(* Logix 5000 project; controller ABB_Drive_Test vendor 1 type 14 code 149 rev 33.12; software revision 33.01; part 5 of 6 *)
(* tags used below, declared in another part *)
   ad_pointer : DINT;
   cf_bigWcmd01 : DINT;
   cf_bigWoffset01 : DINT;
   cfbw01 : CF_big_write;
   check_log_age : BOOL;
   d1hf_copy : BOOL;
   DataIndex : DINT;
   dayms_frac : REAL;
   daysince1900 : DINT;
   daysinprevmonths : DINT[13];
   detect_1st_half_full : BOOL;
   filename : STRING;
   filename_end : STRING;
   filenamestart : STRING;
   ldt : DateTime;
   log_check_active : BOOL;
   logfile_size : DINT;
   logging_enabled : BOOL;   // HABILITAR DATALOGGER
   logpulse : BOOL;
   max_file_size : DINT;
   max_logfiles : DINT;
   nr_of_writes : DINT;
   sec_pulse : TIMER;
   tempstring : STRING;
   tmpDINT : DINT;
   trigger_write : BOOL;
   write_1st_half : BOOL;
   write_length : DINT;
   write_offset : DINT;
   wrSEQ : DINT;
   Year_1901 : DINT;
   asciidata : SINT[11000];
   CF_RW_functions : CF_functions;
   manual_log_trigger : BOOL;
   SrcData : REAL[10];
(* CSVProgram, continued *)

ROUTINE MainRoutine   (* ladder *)
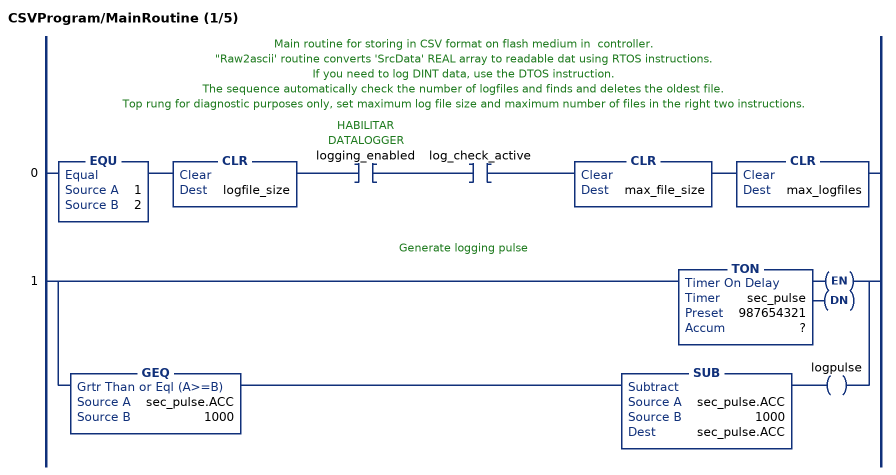
   // Main routine for storing in CSV format on flash medium in  controller.
   // "Raw2ascii' routine converts 'SrcData' REAL array to readable dat using RTOS instructions.
   // If you need to log DINT data, use the DTOS instruction.
   // The sequence automatically check the number of logfiles and finds and deletes the oldest file.
   // Top rung for diagnostic purposes only, set maximum log file size and maximum number of files in the right two instructions.
   0: EQU(1,2)CLR(logfile_size)XIC(logging_enabled)XIC(log_check_active)CLR(max_file_size)CLR(max_logfiles);
   // Generate logging pulse
   1: [TON(sec_pulse,?,?) ,GEQ(sec_pulse.ACC,1000) SUB(sec_pulse.ACC,1000,sec_pulse.ACC) OTE(logpulse) ];
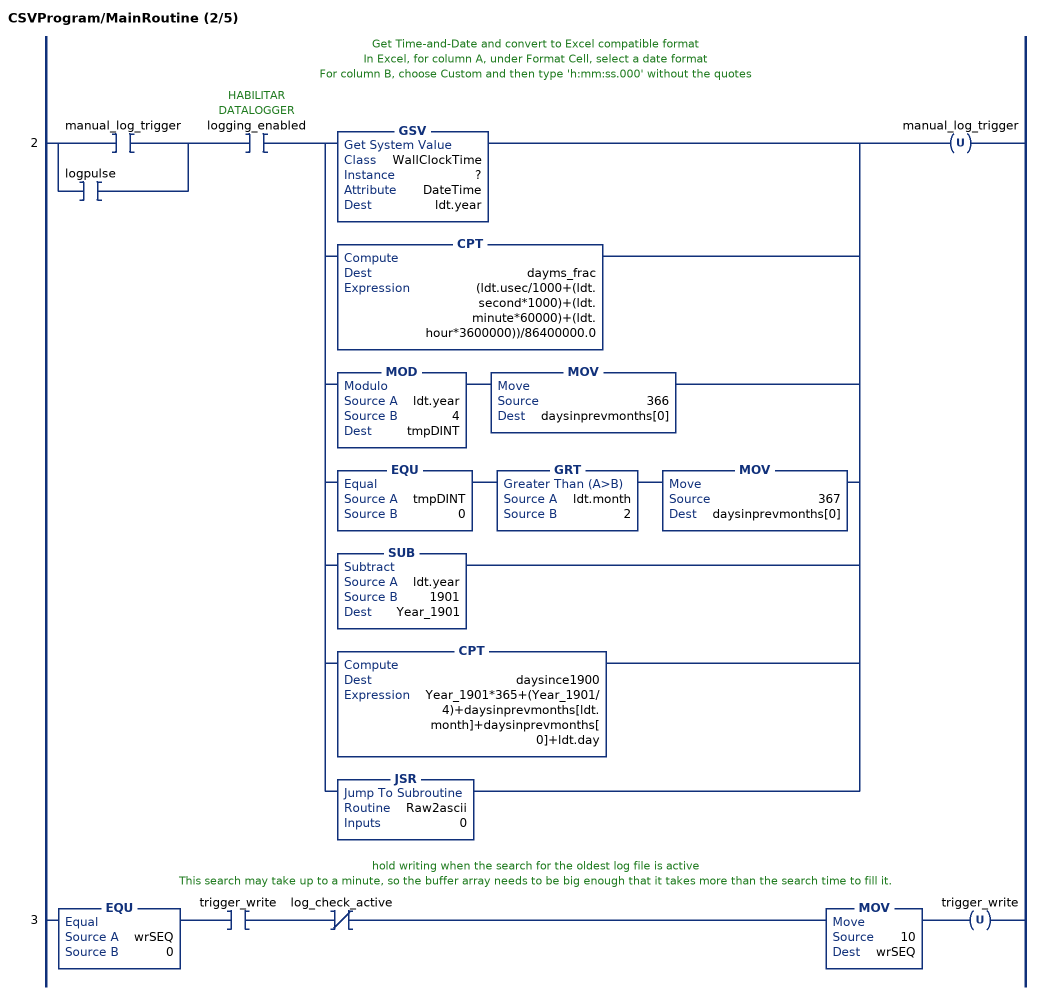
   // Get Time-and-Date and convert to Excel compatible format
   // In Excel, for column A, under Format Cell, select a date format
   // For column B, choose Custom and then type 'h:mm:ss.000' without the quotes
   2: [XIC(manual_log_trigger) ,XIC(logpulse) ]XIC(logging_enabled)[GSV(WallClockTime,?,DateTime,ldt.year) ,CPT(dayms_frac,(ldt.usec/1000+(ldt.second*1000)+(ldt.minute*60000)+(ldt.hour*3600000))/86400000.0) ,MOD(ldt.year,4,tmpDINT) MOV(366,daysinprevmonths[0]) ,EQU(tmpDINT,0) GRT(ldt.month,2) MOV(367,daysinprevmonths[0]) ,SUB(ldt.year,1901,Year_1901) ,CPT(daysince1900,Year_1901*365+(Year_1901/4)+daysinprevmonths[ldt.month]+daysinprevmonths[0]+ldt.day) ,JSR(Raw2ascii,0) ]OTU(manual_log_trigger);
   // hold writing when the search for the oldest log file is active
   // This search may take up to a minute, so the buffer array needs to be big enough that it takes more than the search time to fill it.
   3: EQU(wrSEQ,0)XIC(trigger_write)XIO(log_check_active)MOV(10,wrSEQ)OTU(trigger_write);
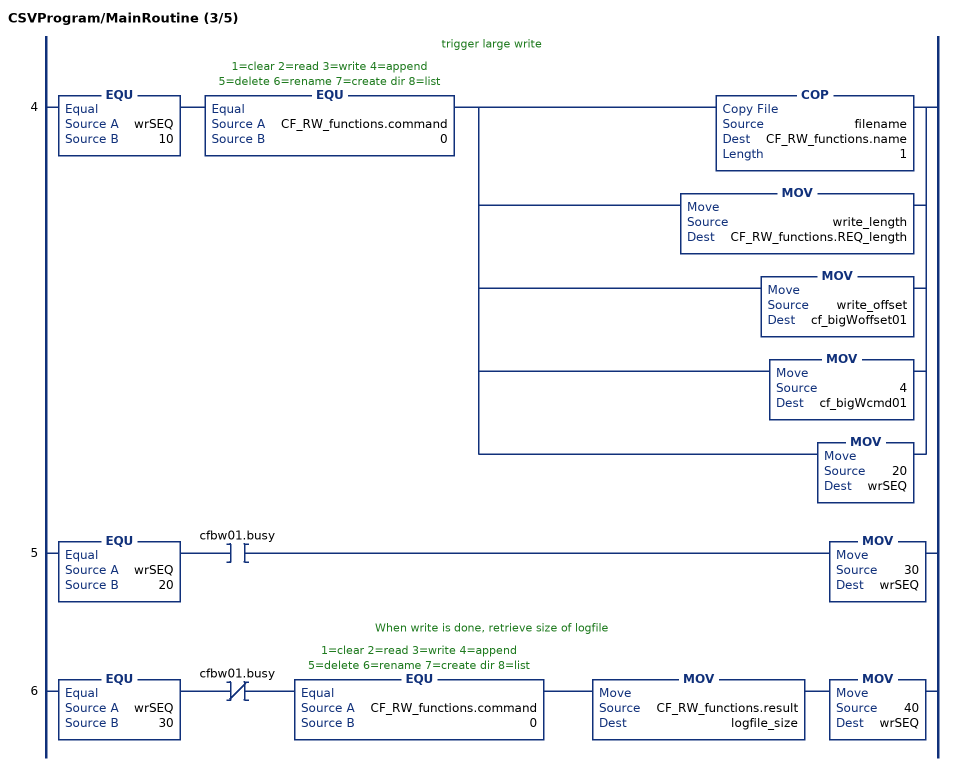
   // trigger large write
   4: EQU(wrSEQ,10)EQU(CF_RW_functions.command,0)[COP(filename,CF_RW_functions.name,1) ,MOV(write_length,CF_RW_functions.REQ_length) ,MOV(write_offset,cf_bigWoffset01) ,MOV(4,cf_bigWcmd01) ,MOV(20,wrSEQ) ];
   5: EQU(wrSEQ,20)XIC(cfbw01.busy)MOV(30,wrSEQ);
   // When write is done, retrieve size of logfile
   6: EQU(wrSEQ,30)XIO(cfbw01.busy)EQU(CF_RW_functions.command,0)MOV(CF_RW_functions.result,logfile_size)MOV(40,wrSEQ);
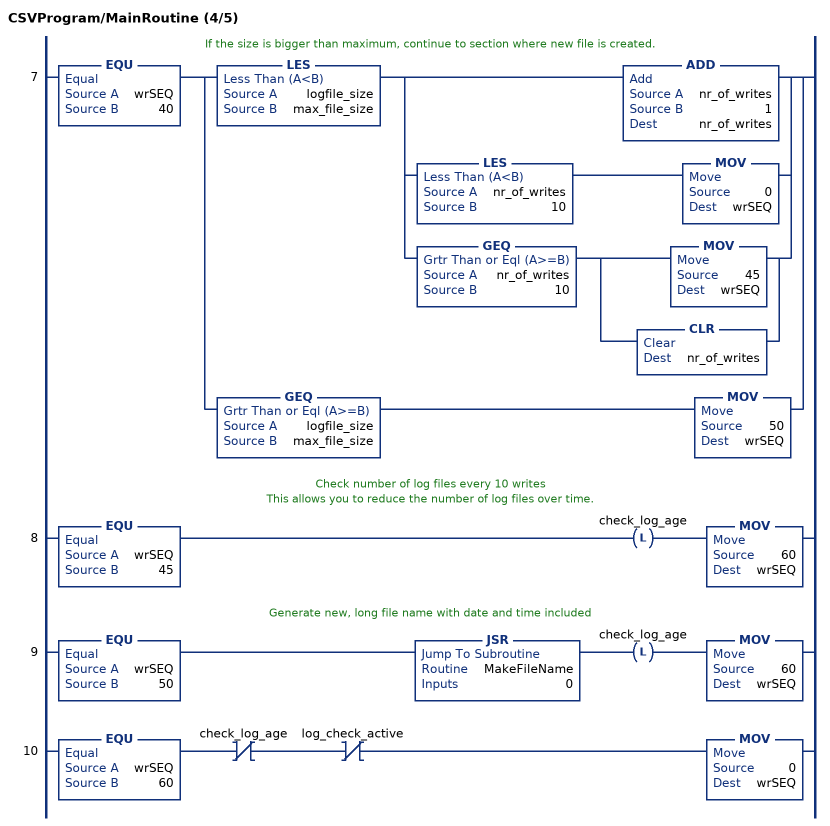
   // If the size is bigger than maximum, continue to section where new file is created.
   7: EQU(wrSEQ,40)[LES(logfile_size,max_file_size) [ADD(nr_of_writes,1,nr_of_writes) ,LES(nr_of_writes,10) MOV(0,wrSEQ) ,GEQ(nr_of_writes,10) [MOV(45,wrSEQ) ,CLR(nr_of_writes) ] ] ,GEQ(logfile_size,max_file_size) MOV(50,wrSEQ) ];
   // Check number of log files every 10 writes
   // This allows you to reduce the number of log files over time.
   8: EQU(wrSEQ,45)OTL(check_log_age)MOV(60,wrSEQ);
   // Generate new, long file name with date and time included
   9: EQU(wrSEQ,50)JSR(MakeFileName,0)OTL(check_log_age)MOV(60,wrSEQ);
   10: EQU(wrSEQ,60)XIO(check_log_age)XIO(log_check_active)MOV(0,wrSEQ);
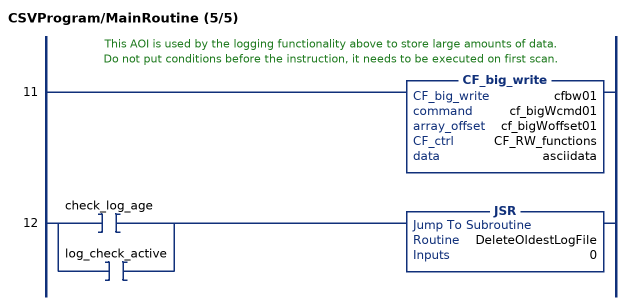
   // This AOI is used by the logging functionality above to store large amounts of data.
   // Do not put conditions before the instruction, it needs to be executed on first scan.
   11: CF_big_write(cfbw01,cf_bigWcmd01,cf_bigWoffset01,CF_RW_functions,asciidata);
   12: [XIC(check_log_age) ,XIC(log_check_active) ]JSR(DeleteOldestLogFile,0);
END_ROUTINE

ROUTINE MakeFileName   (* ladder *)
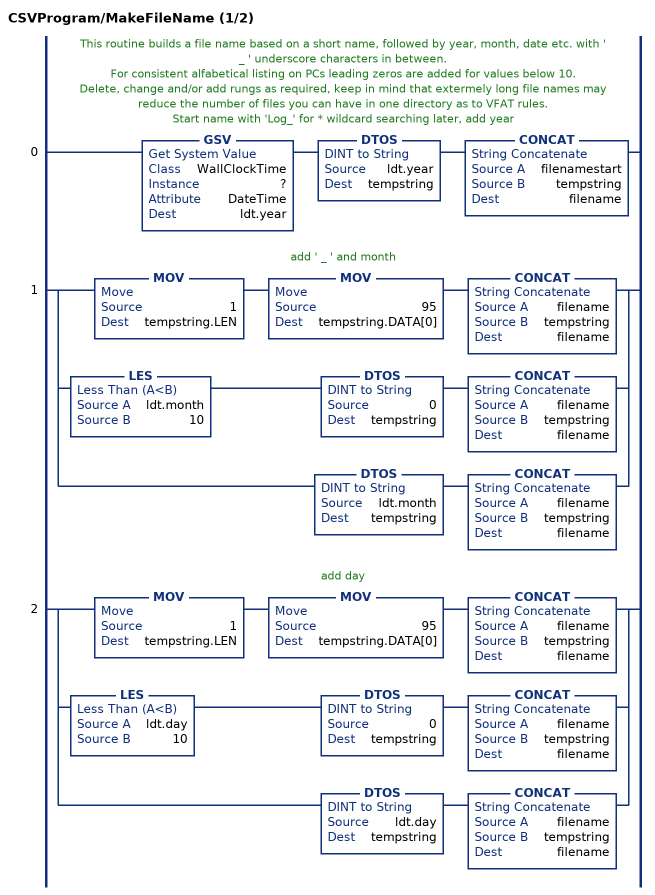
   // This routine builds a file name based on a short name, followed by year, month, date etc. with ' _ ' underscore characters in between.
   // For consistent alfabetical listing on PCs leading zeros are added for values below 10.
   // Delete, change and/or add rungs as required, keep in mind that extermely long file names may reduce the number of files you can have in one directory as to VFAT rules.
   //  Start name with 'Log_' for * wildcard searching later, add year
   0: GSV(WallClockTime,?,DateTime,ldt.year)DTOS(ldt.year,tempstring)CONCAT(filenamestart,tempstring,filename);
   // add ' _ ' and month
   1: [MOV(1,tempstring.LEN) MOV(95,tempstring.DATA[0]) CONCAT(filename,tempstring,filename) ,LES(ldt.month,10) DTOS(0,tempstring) CONCAT(filename,tempstring,filename) ,DTOS(ldt.month,tempstring) CONCAT(filename,tempstring,filename) ];
   // add day
   2: [MOV(1,tempstring.LEN) MOV(95,tempstring.DATA[0]) CONCAT(filename,tempstring,filename) ,LES(ldt.day,10) DTOS(0,tempstring) CONCAT(filename,tempstring,filename) ,DTOS(ldt.day,tempstring) CONCAT(filename,tempstring,filename) ];
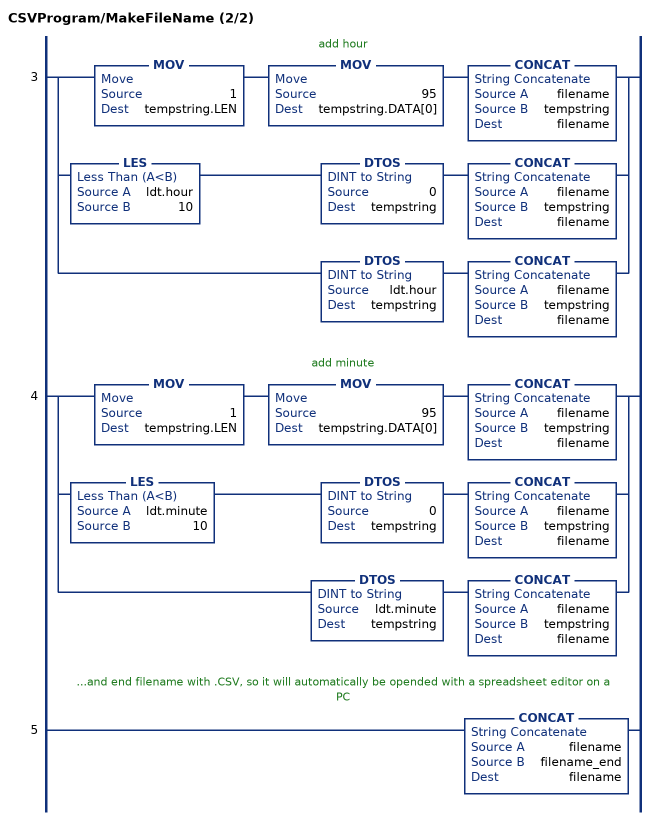
   // add hour
   3: [MOV(1,tempstring.LEN) MOV(95,tempstring.DATA[0]) CONCAT(filename,tempstring,filename) ,LES(ldt.hour,10) DTOS(0,tempstring) CONCAT(filename,tempstring,filename) ,DTOS(ldt.hour,tempstring) CONCAT(filename,tempstring,filename) ];
   // add minute
   4: [MOV(1,tempstring.LEN) MOV(95,tempstring.DATA[0]) CONCAT(filename,tempstring,filename) ,LES(ldt.minute,10) DTOS(0,tempstring) CONCAT(filename,tempstring,filename) ,DTOS(ldt.minute,tempstring) CONCAT(filename,tempstring,filename) ];
   // ...and end filename with .CSV, so it will automatically be opended with a spreadsheet editor on a PC
   5: CONCAT(filename,filename_end,filename);
END_ROUTINE

ROUTINE Raw2ascii   (* structured text *)
   DTOS(daysince1900,tempstring);												//add date in excel compatible format
   tempstring.DATA[tempstring.LEN]:=44;										//add comma
   tempstring.LEN:=tempstring.LEN+1;
   COP ( tempstring.DATA[0],asciidata[ad_pointer],tempstring.LEN);
   ad_pointer:=ad_pointer+tempstring.LEN;
   RTOS(dayms_frac,tempstring);												//add time in excel compatible format
   tempstring.DATA[tempstring.LEN]:=44;										//add comma
   tempstring.LEN:=tempstring.LEN+1;
   COP ( tempstring.DATA[0],asciidata[ad_pointer],tempstring.LEN);
   ad_pointer:=ad_pointer+tempstring.LEN;
   DataIndex:=0;
   For DataIndex := 0 TO 9 DO													//convert array of REALs to asscii
   	RTOS(SrcData[DataIndex],tempstring);
   	IF DataIndex<9 THEN
   		tempstring.DATA[tempstring.LEN]:=44;								//add comma
   		tempstring.LEN:=tempstring.LEN+1;
   	ELSE
   		tempstring.DATA[tempstring.LEN]:=13;								//Carriage return
   		tempstring.DATA[tempstring.LEN+1]:=10;								//Line Feed
   		tempstring.LEN:=tempstring.LEN+2;
   	END_IF;
   	COP ( tempstring.DATA[0],asciidata[ad_pointer],tempstring.LEN);
   	ad_pointer:=ad_pointer+tempstring.LEN;
   END_FOR;
   
   detect_1st_half_full:=(ad_pointer > 5000);									//create oneshot when more than 5000 bytes of data are ready
   write_1st_half:=detect_1st_half_full AND NOT d1hf_copy;
   d1hf_copy:=detect_1st_half_full;
   
   IF write_1st_half THEN 														//trigger write of approx. 5000 bytes
   	write_offset:=0;
   	write_length:=ad_pointer;
   	trigger_write:=1;
   END_IF;
   
   IF ad_pointer > 10000 THEN 													//trigger write of remaining data
   	write_offset:=write_length;
   	write_length:=ad_pointer-write_offset;
   	ad_pointer:=0;
   	trigger_write:=1;
   END_IF;
   
END_ROUTINE
END_PROGRAM

PROGRAM T000_MainProgram   (* main routine R00_MainRoutine *)
VAR
   Acell : BOOL;
   DesAcell : BOOL;
   flagDesAcell : BOOL;   // Flag Auxiliar Boton de Parada
   indiceLocal : DINT;
   InicioDinagram : BOOL;   // Inicio de la Adquisión del Dinagrama
   numeroMuestras : DINT := 280;   // Numero de Muestras del Stroke
   pausa : BOOL;
   rpmFeedback : INT;   // Valor absoluto de la referencia 0 no lo toma
   SCL_01 : SCALE := (In := 3200.0, InRawMax := 19987.0, InRawMin := 3994.0, InEUMax := 20.0, InEUMin := 4.0, Out := 3.2056525, MinAlarm := 1);
   SCL_02 : SCALE := (In := 8894.0, InRawMax := 19987.0, InRawMin := 3994.0, InEUMax := 20.0, InEUMin := 4.0, Out := 8.902144);
   SCL_03 : SCALE := (In := 4045.0, InRawMax := 19987.0, InRawMin := 3994.0, InEUMax := 20.0, InEUMin := 4.0, Out := 4.0510225);
   SCL_04 : SCALE := (In := 4005.0, InRawMax := 19987.0, InRawMin := 3994.0, InEUMax := 20.0, InEUMin := 4.0, Out := 4.011005);
   VCarga : REAL[1500] := ([0] := 11.827799, [1] := 9.4196205, [2] := 9.745639, [3] := 9.745639, [4] := 9.7696495, [5] := 9.7696495, [6] := 9.7696495, [7] := 9.791034, [8] := 9.791034, [9] := 9.770024, [10] := 9.770024, [11] := 9.770024, [12] := 9.797411, [13] := 9.797411, [14] := 9.797411, [15] := 9.822172, [16] := 9.822172, [17] := 9.95573, [18] := 9.95573, [19] := 9.95573, [20] := 9.701369, [21] := 9.701369, [22] := 9.470268, [23] := 9.470268, [24] := 9.470268, [25] := 9.291315, [26] := 9.291315, [27] := 9.291315, [28] := 9.069968, [29] := 9.069968, [30] := 8.960045, [31] := 8.960045, [32] := 8.960045, [33] := 9.023447, [34] := 9.023447, [35] := 9.023447, [36] := 9.019321, [37] := 9.019321, [38] := 8.883512, [39] := 8.883512, [40] := 8.883512, [41] := 8.923655, [42] := 8.923655, [43] := 8.9439125, [44] := 8.9439125, [45] := 8.9439125, [46] := 9.030201, [47] := 9.030201, [48] := 9.030201, [49] := 9.299568, [50] := 9.299568, [51] := 9.464266, [52] := 9.464266, [53] := 9.464266, [54] := 9.457138, [55] := 9.457138, [56] := 9.457138, [57] := 9.626711, [58] := 9.626711, [59] := 9.662352,
        [60] := 9.662352, [61] := 9.662352, [62] := 9.386231, [63] := 9.386231, [64] := 9.347965, [65] := 9.347965, [66] := 9.347965, [67] := 9.220409, [68] := 9.220409, [69] := 8.902645, [70] := 8.902645, [71] := 8.902645, [72] := 8.647533, [73] := 8.647533, [74] := 8.647533, [75] := 8.376289, [76] := 8.376289, [77] := 7.6285872, [78] := 7.6285872, [79] := 7.6285872, [80] := 7.4822736, [81] := 7.4822736, [82] := 7.259051, [83] := 7.259051, [84] := 7.259051, [85] := 7.026449, [86] := 7.026449, [87] := 7.026449, [88] := 6.740574, [89] := 6.740574, [90] := 6.4952164, [91] := 6.4952164, [92] := 6.4952164, [93] := 6.2438564, [94] := 6.2438564, [95] := 6.2438564, [96] := 6.0326395, [97] := 6.0326395, [98] := 6.2190957, [99] := 6.2190957, [100] := 6.2190957, [101] := 6.583005, [102] := 6.583005, [103] := 6.583005, [104] := 6.8467455, [105] := 6.8467455, [106] := 7.3659725, [107] := 7.3659725, [108] := 7.3659725, [109] := 7.469143, [110] := 7.469143, [111] := 7.496905, [112] := 7.496905, [113] := 7.496905, [114] := 7.8848248, [115] := 7.8848248, [116] := 7.8848248, [117] := 7.924967, [118] := 7.924967, [119] := 8.158319,
        [120] := 8.158319, [121] := 8.158319, [122] := 8.3444, [123] := 8.3444, [124] := 8.442694, [125] := 8.442694, [126] := 8.442694, [127] := 8.42356, [128] := 8.42356, [129] := 8.42356, [130] := 8.315514, [131] := 8.315514, [132] := 7.9606075, [133] := 7.9606075, [134] := 7.9606075, [135] := 8.07766, [136] := 8.07766, [137] := 8.042394, [138] := 8.042394, [139] := 8.042394, [140] := 8.178578, [141] := 8.178578, [142] := 8.178578, [143] := 8.174827, [144] := 8.174827, [145] := 8.139561, [146] := 8.139561, [147] := 8.139561, [148] := 8.19471, [149] := 8.19471, [150] := 8.19471, [151] := 8.202964, [152] := 8.202964, [153] := 8.3995495, [154] := 8.3995495, [155] := 8.3995495, [156] := 8.592759, [157] := 8.592759, [158] := 8.938286, [159] := 8.938286, [160] := 8.938286, [161] := 9.0091915, [162] := 9.0091915, [163] := 9.0091915, [164] := 9.1281185, [165] := 9.1281185, [166] := 9.196023, [167] := 9.196023, [168] := 9.196023, [169] := 9.338961, [170] := 9.338961, [171] := 9.480398, [172] := 9.480398, [173] := 9.480398, [174] := 9.461639, [175] := 9.461639, [176] := 9.461639, [177] := 9.607954, [178] := 9.607954, [179] := 9.53217,
        [180] := 9.53217, [181] := 9.53217, [182] := 9.457513, [183] := 9.457513, [184] := 9.457513, [185] := 9.393735, [186] := 9.393735, [187] := 9.398987, [188] := 9.398987, [189] := 9.398987, [190] := 10.072031, [191] := 10.072031, [192] := 10.460326, [193] := 10.460326, [194] := 10.460326, [195] := 10.616395, [196] := 10.616395, [197] := 10.616395, [198] := 10.90452, [199] := 10.90452, [200] := 11.071468, [201] := 11.071468, [202] := 11.071468, [203] := 11.378353, [204] := 11.378353, [205] := 11.463515, [206] := 11.463515, [207] := 11.463515, [208] := 11.71375, [209] := 11.71375, [210] := 11.71375, [211] := 11.889702, [212] := 11.889702, [213] := 11.926468, [214] := 11.926468, [215] := 11.926468, [216] := 11.70362, [217] := 11.70362, [218] := 11.70362, [219] := 11.458638, [220] := 11.458638, [221] := 11.006565, [222] := 11.006565, [223] := 11.006565, [224] := 10.84712, [225] := 10.84712, [226] := 10.508347, [227] := 10.508347, [228] := 10.508347, [229] := 10.232226, [230] := 10.232226, [231] := 10.232226, [232] := 10.07991, [233] := 10.07991, [234] := 9.844307, [235] := 9.844307, [236] := 9.844307, [237] := 9.705121, [238] := 9.705121, [239] := 9.43988,
        [240] := 9.43988, [241] := 9.43988, [242] := 9.398236, [243] := 9.398236, [244] := 9.398236, [245] := 9.730632, [246] := 9.730632, [247] := 9.962858, [248] := 9.962858, [249] := 9.962858, [250] := 10.073156, [251] := 10.073156, [252] := 10.073156, [253] := 10.247232, [254] := 10.247232, [255] := 10.271619, [256] := 10.271619, [257] := 10.271619, [258] := 10.34215, [259] := 10.34215, [260] := 10.348152, [261] := 10.348152, [262] := 10.348152, [263] := 10.3391485, [264] := 10.3391485, [265] := 10.3391485, [266] := 10.533859, [267] := 10.533859, [268] := 10.50272, [269] := 10.50272, [270] := 10.50272, [271] := 10.088914, [272] := 10.088914, [273] := 9.71525, [274] := 9.71525, [275] := 9.71525, [276] := 9.600075, [277] := 9.600075, [278] := 9.600075, [279] := 9.190395, [280] := 9.190395, [281] := 9.1281185, [282] := 9.1281185, [283] := 9.1281185, [284] := 9.05121, [285] := 9.05121, [286] := 8.89139, [287] := 8.89139, [288] := 8.89139, [289] := 8.768711, [290] := 8.768711, [291] := 8.768711, [292] := 8.70756, [293] := 8.70756, [294] := 8.6021385, [295] := 8.6021385, [296] := 8.6021385, [297] := 8.784093, [298] := 8.784093, [299] := 9.2219095,
        [300] := 9.2219095, [301] := 9.2219095, [302] := 9.306322, [303] := 9.306322, [304] := 9.306322, [305] := 9.615831, [306] := 9.615831, [307] := 9.742262, [308] := 9.742262, [309] := 9.742262, [310] := 9.7797785, [311] := 9.7797785, [312] := 9.791034, [313] := 9.791034, [314] := 9.791034, [315] := 9.77265, [316] := 9.77265, [317] := 9.77265, [318] := 9.82855, [319] := 9.82855, [320] := 9.89758, [321] := 9.89758, [322] := 9.89758, [323] := 9.8266735, [324] := 9.8266735, [325] := 9.590696, [326] := 9.590696, [327] := 9.590696, [328] := 9.310073, [329] := 9.310073, [330] := 9.310073, [331] := 9.281185, [332] := 9.281185, [333] := 9.080097, [334] := 9.080097, [335] := 9.080097, [336] := 8.944663, [337] := 8.944663, [338] := 9.016695, [339] := 9.016695, [340] := 9.016695, [341] := 8.874883, [342] := 8.874883, [343] := 8.874883, [344] := 8.983305, [345] := 8.983305, [346] := 8.969799, [347] := 8.969799, [348] := 8.969799, [349] := 8.959295, [350] := 8.959295, [351] := 9.151753, [352] := 9.151753, [353] := 9.151753, [354] := 9.517163, [355] := 9.517163, [356] := 9.517163, [357] := 9.475145, [358] := 9.475145, [359] := 9.5820675,
        [360] := 9.5820675, [361] := 9.5820675, [362] := 9.595948, [363] := 9.595948, [364] := 9.453011, [365] := 9.453011, [366] := 9.453011, [367] := 9.394485, [368] := 9.394485, [369] := 9.394485, [370] := 9.338961, [371] := 9.338961, [372] := 9.012193, [373] := 9.012193, [374] := 9.012193, [375] := 8.838491, [376] := 8.838491, [377] := 8.425061, [378] := 8.425061, [379] := 8.425061, [380] := 7.739636, [381] := 7.739636, [382] := 7.739636, [383] := 7.4897766, [384] := 7.4897766, [385] := 7.2721815, [386] := 7.2721815, [387] := 7.2721815, [388] := 7.059088, [389] := 7.059088, [390] := 6.730069, [391] := 6.730069, [392] := 6.730069, [393] := 6.590133, [394] := 6.590133, [395] := 6.590133, [396] := 6.438192, [397] := 6.438192, [398] := 6.066779, [399] := 6.066779, [400] := 6.066779, [401] := 6.139561, [402] := 6.139561, [403] := 6.139561, [404] := 6.4865875, [405] := 6.4865875, [406] := 7.0208216, [407] := 7.0208216, [408] := 7.0208216, [409] := 7.308573, [410] := 7.308573, [411] := 7.4695177, [412] := 7.4695177, [413] := 7.4695177, [414] := 7.4646406, [415] := 7.4646406, [416] := 7.8806977, [417] := 7.8806977, [418] := 7.8806977, [419] := 7.935847,
        [420] := 7.935847, [421] := 7.935847, [422] := 8.08141, [423] := 8.08141, [424] := 8.407804, [425] := 8.407804, [426] := 8.407804, [427] := 8.448321, [428] := 8.448321, [429] := 8.448321, [430] := 8.42356, [431] := 8.42356, [432] := 8.313262, [433] := 8.313262, [434] := 8.313262, [435] := 7.9673605, [436] := 7.9673605, [437] := 8.078033, [438] := 8.078033, [439] := 8.078033, [440] := 8.042394, [441] := 8.042394, [442] := 8.042394, [443] := 8.150065, [444] := 8.150065, [445] := 8.199963, [446] := 8.199963, [447] := 8.199963, [448] := 8.118176, [449] := 8.118176, [450] := 8.21797, [451] := 8.21797, [452] := 8.21797, [453] := 8.210467, [454] := 8.210467, [455] := 8.401051, [456] := 8.401051, [457] := 8.401051, [458] := 8.592759, [459] := 8.592759, [460] := 8.592759, [461] := 8.931908, [462] := 8.931908, [463] := 9.018946, [464] := 9.018946, [465] := 9.018946, [466] := 9.132245, [467] := 9.132245, [468] := 9.132245, [469] := 9.229413, [470] := 9.229413, [471] := 9.411742, [472] := 9.411742, [473] := 9.411742, [474] := 9.468018, [475] := 9.468018, [476] := 9.499531, [477] := 9.499531, [478] := 9.499531, [479] := 9.555056,
        [480] := 9.555056, [481] := 9.555056, [482] := 9.484524, [483] := 9.484524, [484] := 9.468392, [485] := 9.468392, [486] := 9.468392, [487] := 9.367848, [488] := 9.367848, [489] := 9.367848, [490] := 9.56481, [491] := 9.56481, [492] := 10.21797, [493] := 10.21797, [494] := 10.21797, [495] := 10.521478, [496] := 10.521478, [497] := 10.678296, [498] := 10.678296, [499] := 10.678296, [500] := 10.929657, [501] := 10.929657, [502] := 10.929657, [503] := 11.0845995, [504] := 11.0845995, [505] := 11.428249, [506] := 11.428249, [507] := 11.428249, [508] := 11.508909, [509] := 11.508909, [510] := 11.779404, [511] := 11.779404, [512] := 11.779404, [513] := 11.864941, [514] := 11.864941, [515] := 11.864941, [516] := 11.923092, [517] := 11.923092, [518] := 11.53367, [519] := 11.53367, [520] := 11.53367, [521] := 11.324329, [522] := 11.324329, [523] := 10.936409, [524] := 10.936409, [525] := 10.936409, [526] := 10.784468, [527] := 10.784468, [528] := 10.784468, [529] := 10.437441, [530] := 10.437441, [531] := 10.18308, [532] := 10.18308, [533] := 10.18308, [534] := 10.073532, [535] := 10.073532, [536] := 9.767774, [537] := 9.767774, [538] := 9.767774, [539] := 9.62446,
        [540] := 9.62446, [541] := 9.62446, [542] := 9.457138, [543] := 9.457138, [544] := 9.595948, [545] := 9.595948, [546] := 9.595948, [547] := 9.763646, [548] := 9.763646, [549] := 9.763646, [550] := 9.963984, [551] := 9.963984, [552] := 10.061527, [553] := 10.061527, [554] := 10.061527, [555] := 10.22885, [556] := 10.22885, [557] := 10.250235, [558] := 10.250235, [559] := 10.250235, [560] := 10.329019, [561] := 10.329019, [562] := 10.329019, [563] := 10.365034, [564] := 10.365034, [565] := 10.3642845, [566] := 10.3642845, [567] := 10.3642845, [568] := 10.548115, [569] := 10.548115, [570] := 10.568374, [571] := 10.568374, [572] := 10.568374, [573] := 10.117051, [574] := 10.117051, [575] := 10.117051, [576] := 9.7512665, [577] := 9.7512665, [578] := 9.630088, [579] := 9.630088, [580] := 9.630088, [581] := 9.216658, [582] := 9.216658, [583] := 9.134121, [584] := 9.134121, [585] := 9.134121, [586] := 9.048584, [587] := 9.048584, [588] := 9.048584, [589] := 8.772087, [590] := 8.772087, [591] := 8.723316, [592] := 8.723316, [593] := 8.723316, [594] := 8.709061, [595] := 8.709061, [596] := 8.709061, [597] := 8.557118, [598] := 8.557118, [599] := 8.752579,
        [600] := 8.752579, [601] := 8.752579, [602] := 9.01857, [603] := 9.01857, [604] := 9.305946, [605] := 9.305946, [606] := 9.305946, [607] := 9.6038265, [608] := 9.6038265, [609] := 9.6038265, [610] := 9.744513, [611] := 9.744513, [612] := 9.780153, [613] := 9.780153, [614] := 9.780153, [615] := 9.7797785, [616] := 9.7797785, [617] := 9.80604, [618] := 9.80604, [619] := 9.80604, [620] := 9.804164, [621] := 9.804164, [622] := 9.804164, [623] := 9.896455, [624] := 9.896455, [625] := 9.867191, [626] := 9.867191, [627] := 9.867191, [628] := 9.549052, [629] := 9.549052, [630] := 9.310448, [631] := 9.310448, [632] := 9.310448, [633] := 9.236166, [634] := 9.236166, [635] := 9.06509, [636] := 9.06509, [637] := 9.06509, [638] := 8.968674, [639] := 8.968674, [640] := 8.968674, [641] := 9.052711, [642] := 9.052711, [643] := 8.884637, [644] := 8.884637, [645] := 8.884637, [646] := 8.908648, [647] := 8.908648, [648] := 8.908648, [649] := 8.944288, [650] := 8.944288, [651] := 8.920278, [652] := 8.920278, [653] := 8.920278, [654] := 9.137122, [655] := 9.137122, [656] := 9.485649, [657] := 9.485649, [658] := 9.485649, [659] := 9.455637,
        [660] := 9.455637, [661] := 9.455637, [662] := 9.576815, [663] := 9.576815, [664] := 9.630088, [665] := 9.630088, [666] := 9.630088, [667] := 9.455637, [668] := 9.455637, [669] := 9.395235, [670] := 9.395235, [671] := 9.395235, [672] := 9.342337, [673] := 9.342337, [674] := 9.342337, [675] := 9.020447, [676] := 9.020447, [677] := 8.723316, [678] := 8.723316, [679] := 8.723316, [680] := 8.434814, [681] := 8.434814, [682] := 7.8825736, [683] := 7.8825736, [684] := 7.8825736, [685] := 7.574939, [686] := 7.574939, [687] := 7.574939, [688] := 7.3453383, [689] := 7.3453383, [690] := 7.202401, [691] := 7.202401, [692] := 7.202401, [693] := 7.202401, [694] := 6.470831, [695] := 6.2318516, [696] := 6.1268053, [697] := 6.1283064, [698] := 6.2566123, [699] := 6.5015945, [700] := 6.829488, [701] := 7.2567997, [702] := 7.5719376, [703] := 8.032264, [704] := 8.511349, [705] := 8.931157, [706] := 9.431252, [707] := 9.95348, [708] := 10.449821, [709] := 10.877884, [710] := 11.1885195, [711] := 11.550178, [712] := 11.802288, [713] := 11.975239, [714] := 12.04577, [715] := 12.064903, [716] := 12.011254, [717] := 11.886701, [718] := 11.722754, [719] := 11.55468,
        [720] := 11.320202, [721] := 11.037329, [722] := 10.713187, [723] := 10.439317, [724] := 10.081785, [725] := 9.656725, [726] := 9.211781, [727] := 8.746576, [728] := 8.394298, [729] := 7.8938284, [730] := 7.385481, [731] := 7.0384545, [732] := 6.6576624, [733] := 6.37704, [734] := 6.25061, [735] := 6.135434, [736] := 6.132808, [737] := 6.2322264, [738] := 6.4569497, [739] := 6.781467, [740] := 7.156631, [741] := 7.580191, [742] := 7.9636087, [743] := 8.440818, [744] := 8.94879, [745] := 9.467642, [746] := 9.989495, [747] := 10.374788, [748] := 10.827987, [749] := 11.235415, [750] := 11.583942, [751] := 11.786907, [752] := 11.959857, [753] := 12.050648, [754] := 12.062277, [755] := 12.019883, [756] := 11.9020815, [757] := 11.734009, [758] := 11.524292, [759] := 11.287188, [760] := 11.042206, [761] := 10.725567, [762] := 10.368411, [763] := 9.978615, [764] := 9.63459, [765] := 9.160382, [766] := 8.693303, [767] := 8.187207, [768] := 7.703245, [769] := 7.3678484, [770] := 6.9619207, [771] := 6.610392, [772] := 6.3822923, [773] := 6.1935844, [774] := 6.1204276, [775] := 6.166948, [776] := 6.2453575, [777] := 6.5045958, [778] := 6.717689, [779] := 7.077096,
        [780] := 7.525042, [781] := 7.968111, [782] := 8.438566, [783] := 8.844494, [784] := 9.386982, [785] := 9.897205, [786] := 10.383793, [787] := 10.742825, [788] := 11.151003, [789] := 11.49878, [790] := 11.775652, [791] := 11.959482, [792] := 12.040893, [793] := 12.066403, [794] := 12.021384, [795] := 11.910336, [796] := 11.785781, [797] := 11.588445, [798] := 11.33746, [799] := 11.060964, [800] := 11.060964);
   Vct : REAL[1500];
   VPosicion : REAL[1500] := ([1] := 100.981674, [2] := 101.10048, [3] := 101.10048, [4] := 101.14424, [5] := 101.14424, [6] := 101.14424, [7] := 101.10048, [8] := 101.10048, [9] := 100.88164, [10] := 100.88164, [11] := 100.88164, [12] := 100.694046, [13] := 100.694046, [14] := 100.694046, [15] := 100.13131, [16] := 100.13131, [17] := 99.49977, [18] := 99.49977, [19] := 99.49977, [20] := 99.0871, [21] := 99.0871, [22] := 98.167946, [23] := 98.167946, [24] := 98.167946, [25] := 97.07997, [26] := 97.07997, [27] := 97.07997, [28] := 96.504715, [29] := 96.504715, [30] := 95.61683, [31] := 95.61683, [32] := 95.61683, [33] := 94.92903, [34] := 94.92903, [35] := 94.92903, [36] := 93.45963, [37] := 93.45963, [38] := 92.728065, [39] := 92.728065, [40] := 92.728065, [41] := 91.13986, [42] := 91.13986, [43] := 89.32033, [44] := 89.32033, [45] := 89.32033, [46] := 88.407425, [47] := 88.407425, [48] := 88.407425, [49] := 86.46908, [50] := 86.46908, [51] := 85.43112, [52] := 85.43112, [53] := 85.43112, [54] := 83.35521, [55] := 83.35521, [56] := 83.35521, [57] := 82.348526, [58] := 82.348526, [59] := 80.20384, [60] := 80.20384,
        [61] := 80.20384, [62] := 77.77777, [63] := 77.77777, [64] := 76.74608, [65] := 76.74608, [66] := 76.74608, [67] := 74.32626, [68] := 74.32626, [69] := 72.40668, [70] := 72.40668, [71] := 72.40668, [72] := 71.05608, [73] := 71.05608, [74] := 71.05608, [75] := 68.51748, [76] := 68.51748, [77] := 66.841736, [78] := 66.841736, [79] := 66.841736, [80] := 64.37816, [81] := 64.37816, [82] := 61.601948, [83] := 61.601948, [84] := 61.601948, [85] := 59.98249, [86] := 59.98249, [87] := 59.98249, [88] := 56.8061, [89] := 56.8061, [90] := 55.29294, [91] := 55.29294, [92] := 55.29294, [93] := 52.085285, [94] := 52.085285, [95] := 52.085285, [96] := 50.434566, [97] := 50.434566, [98] := 47.645844, [99] := 47.645844, [100] := 47.645844, [101] := 44.544483, [102] := 44.544483, [103] := 44.544483, [104] := 42.906273, [105] := 42.906273, [106] := 39.736134, [107] := 39.736134, [108] := 39.736134, [109] := 38.366783, [110] := 38.366783, [111] := 34.821487, [112] := 34.821487, [113] := 34.821487, [114] := 33.16451, [115] := 33.16451, [116] := 33.16451, [117] := 29.87557, [118] := 29.87557, [119] := 26.692926, [120] := 26.692926,
        [121] := 26.692926, [122] := 25.048458, [123] := 25.048458, [124] := 22.209717, [125] := 22.209717, [126] := 22.209717, [127] := 20.433939, [128] := 20.433939, [129] := 20.433939, [130] := 17.939096, [131] := 17.939096, [132] := 15.031576, [133] := 15.031576, [134] := 15.031576, [135] := 13.449633, [136] := 13.449633, [137] := 11.329955, [138] := 11.329955, [139] := 11.329955, [140] := 9.222785, [141] := 9.222785, [142] := 9.222785, [143] := 8.15982, [144] := 8.15982, [145] := 6.3715367, [146] := 6.3715367, [147] := 6.3715367, [148] := 5.5836916, [149] := 5.5836916, [150] := 5.5836916, [151] := 4.2956295, [152] := 4.2956295, [153] := 3.7516415, [154] := 3.7516415, [155] := 3.7516415, [156] := 2.8449953, [157] := 2.8449953, [158] := 2.3260176, [159] := 2.3260176, [160] := 2.3260176, [161] := 2.1196783, [162] := 2.1196783, [163] := 2.1196783, [164] := 1.9946218, [165] := 1.9946218, [166] := 2.0133793, [167] := 2.0133793, [168] := 2.0133793, [169] := 2.225974, [170] := 2.225974, [171] := 2.5261045, [172] := 2.5261045, [173] := 2.5261045, [174] := 3.3577204, [175] := 3.3577204, [176] := 3.3577204, [177] := 4.63953, [178] := 4.63953, [179] := 5.158508, [180] := 5.158508,
        [181] := 5.158508, [182] := 6.5341086, [183] := 6.5341086, [184] := 6.5341086, [185] := 7.6158314, [186] := 7.6158314, [187] := 9.810543, [188] := 9.810543, [189] := 9.810543, [190] := 11.898955, [191] := 11.898955, [192] := 12.730569, [193] := 12.730569, [194] := 12.730569, [195] := 14.793971, [196] := 14.793971, [197] := 14.793971, [198] := 17.382605, [199] := 17.382605, [200] := 18.651909, [201] := 18.651909, [202] := 18.651909, [203] := 21.334332, [204] := 21.334332, [205] := 22.709936, [206] := 22.709936, [207] := 22.709936, [208] := 25.4799, [209] := 25.4799, [210] := 25.4799, [211] := 27.111864, [212] := 27.111864, [213] := 30.063152, [214] := 30.063152, [215] := 30.063152, [216] := 32.93316, [217] := 32.93316, [218] := 32.93316, [219] := 34.571373, [220] := 34.571373, [221] := 37.99162, [222] := 37.99162, [223] := 37.99162, [224] := 39.81117, [225] := 39.81117, [226] := 43.387733, [227] := 43.387733, [228] := 43.387733, [229] := 45.057213, [230] := 45.057213, [231] := 45.057213, [232] := 48.640026, [233] := 48.640026, [234] := 52.079033, [235] := 52.079033, [236] := 52.079033, [237] := 54.286247, [238] := 54.286247, [239] := 57.706493, [240] := 57.706493,
        [241] := 57.706493, [242] := 59.394733, [243] := 59.394733, [244] := 59.394733, [245] := 62.714935, [246] := 62.714935, [247] := 66.003876, [248] := 66.003876, [249] := 66.003876, [250] := 67.63584, [251] := 67.63584, [252] := 67.63584, [253] := 70.899765, [254] := 70.899765, [255] := 74.15119, [256] := 74.15119, [257] := 74.15119, [258] := 75.82066, [259] := 75.82066, [260] := 78.9658, [261] := 78.9658, [262] := 78.9658, [263] := 80.42893, [264] := 80.42893, [265] := 80.42893, [266] := 82.811226, [267] := 82.811226, [268] := 84.15556, [269] := 84.15556, [270] := 84.15556, [271] := 87.031815, [272] := 87.031815, [273] := 89.3641, [274] := 89.3641, [275] := 89.3641, [276] := 90.28325, [277] := 90.28325, [278] := 90.28325, [279] := 92.43419, [280] := 92.43419, [281] := 93.26579, [282] := 93.26579, [283] := 93.26579, [284] := 94.92278, [285] := 94.92278, [286] := 95.7669, [287] := 95.7669, [288] := 95.7669, [289] := 97.31132, [290] := 97.31132, [291] := 97.31132, [292] := 98.499344, [293] := 98.499344, [294] := 99.03083, [295] := 99.03083, [296] := 99.03083, [297] := 99.88744, [298] := 99.88744, [299] := 100.51272, [300] := 100.51272,
        [301] := 100.51272, [302] := 100.75033, [303] := 100.75033, [304] := 100.75033, [305] := 101.0317, [306] := 101.0317, [307] := 101.14424, [308] := 101.14424, [309] := 101.14424, [310] := 101.12549, [311] := 101.12549, [312] := 101.05046, [313] := 101.05046, [314] := 101.05046, [315] := 100.70655, [316] := 100.70655, [317] := 100.70655, [318] := 100.19383, [319] := 100.19383, [320] := 99.93746, [321] := 99.93746, [322] := 99.93746, [323] := 99.18713, [324] := 99.18713, [325] := 98.78697, [326] := 98.78697, [327] := 98.78697, [328] := 97.84906, [329] := 97.84906, [330] := 97.84906, [331] := 97.38636, [332] := 97.38636, [333] := 96.09203, [334] := 96.09203, [335] := 96.09203, [336] := 94.82899, [337] := 94.82899, [338] := 93.41587, [339] := 93.41587, [340] := 93.41587, [341] := 92.67179, [342] := 92.67179, [343] := 92.67179, [344] := 91.16487, [345] := 91.16487, [346] := 90.364525, [347] := 90.364525, [348] := 90.364525, [349] := 88.63878, [350] := 88.63878, [351] := 87.750885, [352] := 87.750885, [353] := 87.750885, [354] := 85.825035, [355] := 85.825035, [356] := 85.825035, [357] := 83.76164, [358] := 83.76164, [359] := 82.64866, [360] := 82.64866,
        [361] := 82.64866, [362] := 80.71656, [363] := 80.71656, [364] := 79.59732, [365] := 79.59732, [366] := 79.59732, [367] := 76.89614, [368] := 76.89614, [369] := 76.89614, [370] := 75.82692, [371] := 75.82692, [372] := 73.19452, [373] := 73.19452, [374] := 73.19452, [375] := 70.68092, [376] := 70.68092, [377] := 69.63671, [378] := 69.63671, [379] := 69.63671, [380] := 66.9668, [381] := 66.9668, [382] := 66.9668, [383] := 65.71625, [384] := 65.71625, [385] := 62.639904, [386] := 62.639904, [387] := 62.639904, [388] := 61.251797, [389] := 61.251797, [390] := 58.35678, [391] := 58.35678, [392] := 58.35678, [393] := 55.34296, [394] := 55.34296, [395] := 55.34296, [396] := 53.84856, [397] := 53.84856, [398] := 51.272427, [399] := 51.272427, [400] := 51.272427, [401] := 47.75839, [402] := 47.75839, [403] := 47.75839, [404] := 46.151436, [405] := 46.151436, [406] := 42.943787, [407] := 42.943787, [408] := 42.943787, [409] := 41.311825, [410] := 41.311825, [411] := 38.01663, [412] := 38.01663, [413] := 38.01663, [414] := 36.334644, [415] := 36.334644, [416] := 33.12699, [417] := 33.12699, [418] := 33.12699, [419] := 29.444134, [420] := 29.444134,
        [421] := 29.444134, [422] := 28.074783, [423] := 28.074783, [424] := 24.723316, [425] := 24.723316, [426] := 24.723316, [427] := 23.010067, [428] := 23.010067, [429] := 23.010067, [430] := 20.1213, [431] := 20.1213, [432] := 18.72069, [433] := 18.72069, [434] := 18.72069, [435] := 15.950727, [436] := 15.950727, [437] := 13.3308325, [438] := 13.3308325, [439] := 13.3308325, [440] := 10.911024, [441] := 10.911024, [442] := 10.911024, [443] := 9.766772, [444] := 9.766772, [445] := 7.659602, [446] := 7.659602, [447] := 7.659602, [448] := 6.72169, [449] := 6.72169, [450] := 5.077222, [451] := 5.077222, [452] := 5.077222, [453] := 4.545739, [454] := 4.545739, [455] := 3.507784, [456] := 3.507784, [457] := 3.507784, [458] := 2.7074337, [459] := 2.7074337, [460] := 2.7074337, [461] := 2.401051, [462] := 2.401051, [463] := 2.0446448, [464] := 2.0446448, [465] := 2.0446448, [466] := 2.0071268, [467] := 2.0071268, [468] := 2.0071268, [469] := 2.08216, [470] := 2.08216, [471] := 2.213469, [472] := 2.213469, [473] := 2.213469, [474] := 2.888763, [475] := 2.888763, [476] := 3.86419, [477] := 3.86419, [478] := 3.86419, [479] := 4.483211, [480] := 4.483211,
        [481] := 4.483211, [482] := 5.846307, [483] := 5.846307, [484] := 6.715438, [485] := 6.715438, [486] := 6.715438, [487] := 8.4599495, [488] := 8.4599495, [489] := 8.4599495, [490] := 10.517102, [491] := 10.517102, [492] := 11.586321, [493] := 11.586321, [494] := 11.586321, [495] := 13.731009, [496] := 13.731009, [497] := 15.181643, [498] := 15.181643, [499] := 15.181643, [500] := 17.388857, [501] := 17.388857, [502] := 17.388857, [503] := 19.764894, [504] := 19.764894, [505] := 21.496904, [506] := 21.496904, [507] := 21.496904, [508] := 24.648281, [509] := 24.648281, [510] := 26.161444, [511] := 26.161444, [512] := 26.161444, [513] := 29.087723, [514] := 29.087723, [515] := 29.087723, [516] := 30.600887, [517] := 30.600887, [518] := 33.814793, [519] := 33.814793, [520] := 33.814793, [521] := 36.71606, [522] := 36.71606, [523] := 38.279247, [524] := 38.279247, [525] := 38.279247, [526] := 41.468143, [527] := 41.468143, [528] := 41.468143, [529] := 43.06259, [530] := 43.06259, [531] := 46.58288, [532] := 46.58288, [533] := 46.58288, [534] := 49.809288, [535] := 49.809288, [536] := 52.029015, [537] := 52.029015, [538] := 52.029015, [539] := 55.092854, [540] := 55.092854,
        [541] := 55.092854, [542] := 58.000374, [543] := 58.000374, [544] := 60.095043, [545] := 60.095043, [546] := 60.095043, [547] := 63.70912, [548] := 63.70912, [549] := 63.70912, [550] := 65.441124, [551] := 65.441124, [552] := 68.43619, [553] := 68.43619, [554] := 68.43619, [555] := 69.87431, [556] := 69.87431, [557] := 72.73182, [558] := 72.73182, [559] := 72.73182, [560] := 76.17082, [561] := 76.17082, [562] := 76.17082, [563] := 77.290054, [564] := 77.290054, [565] := 80.54149, [566] := 80.54149, [567] := 80.54149, [568] := 81.91708, [569] := 81.91708, [570] := 84.56824, [571] := 84.56824, [572] := 84.56824, [573] := 85.85631, [574] := 85.85631, [575] := 85.85631, [576] := 88.251114, [577] := 88.251114, [578] := 90.41455, [579] := 90.41455, [580] := 90.41455, [581] := 91.71512, [582] := 91.71512, [583] := 93.697235, [584] := 93.697235, [585] := 93.697235, [586] := 95.448006, [587] := 95.448006, [588] := 95.448006, [589] := 96.2296, [590] := 96.2296, [591] := 97.56768, [592] := 97.56768, [593] := 97.56768, [594] := 98.14294, [595] := 98.14294, [596] := 98.14294, [597] := 99.16838, [598] := 99.16838, [599] := 99.612335, [600] := 99.612335,
        [601] := 99.612335, [602] := 100.343895, [603] := 100.343895, [604] := 100.85663, [605] := 100.85663, [606] := 100.85663, [607] := 101.00668, [608] := 101.00668, [609] := 101.00668, [610] := 101.1505, [611] := 101.1505, [612] := 101.14424, [613] := 101.14424, [614] := 101.14424, [615] := 100.981674, [616] := 100.981674, [617] := 100.81285, [618] := 100.81285, [619] := 100.81285, [620] := 100.33139, [621] := 100.33139, [622] := 100.33139, [623] := 99.69361, [624] := 99.69361, [625] := 99.33095, [626] := 99.33095, [627] := 99.33095, [628] := 98.5181, [629] := 98.5181, [630] := 97.68024, [631] := 97.68024, [632] := 97.68024, [633] := 97.01744, [634] := 97.01744, [635] := 95.848175, [636] := 95.848175, [637] := 95.848175, [638] := 95.229164, [639] := 95.229164, [640] := 95.229164, [641] := 93.86606, [642] := 93.86606, [643] := 92.16533, [644] := 92.16533, [645] := 92.16533, [646] := 91.38998, [647] := 91.38998, [648] := 91.38998, [649] := 89.8393, [650] := 89.8393, [651] := 88.87012, [652] := 88.87012, [653] := 88.87012, [654] := 87.09435, [655] := 87.09435, [656] := 86.100174, [657] := 86.100174, [658] := 86.100174, [659] := 84.03676, [660] := 84.03676,
        [661] := 84.03676, [662] := 82.42982, [663] := 82.42982, [664] := 81.32932, [665] := 81.32932, [666] := 81.32932, [667] := 78.8595, [668] := 78.8595, [669] := 77.62146, [670] := 77.62146, [671] := 77.62146, [672] := 75.25168, [673] := 75.25168, [674] := 75.25168, [675] := 74.02613, [676] := 74.02613, [677] := 71.83142, [678] := 71.83142, [679] := 71.83142, [680] := 69.11774, [681] := 69.11774, [682] := 68.09854, [683] := 68.09854, [684] := 68.09854, [685] := 65.31608, [686] := 65.31608, [687] := 65.31608, [688] := 62.533604, [689] := 62.533604, [690] := 61.201775, [691] := 61.201775, [692] := 61.201775, [693] := 61.201775, [694] := 7.847184, [695] := 3.86419, [696] := 2.1134257, [697] := 2.1384358, [698] := 4.2768717, [699] := 8.359906, [700] := 13.824797, [701] := 20.946663, [702] := 26.19896, [703] := 33.871067, [704] := 41.855812, [705] := 48.852623, [706] := 57.187515, [707] := 65.89133, [708] := 74.1637, [709] := 81.298065, [710] := 86.47533, [711] := 92.50296, [712] := 96.7048, [713] := 99.58732, [714] := 100.76283, [715] := 101.08172, [716] := 100.18758, [717] := 98.11168, [718] := 95.379234, [719] := 92.578, [720] := 88.67004,
        [721] := 83.955475, [722] := 78.553116, [723] := 73.98862, [724] := 68.02976, [725] := 60.945408, [726] := 53.529667, [727] := 45.77627, [728] := 39.904957, [729] := 31.563807, [730] := 23.091352, [731] := 17.307573, [732] := 10.961044, [733] := 6.2839985, [734] := 4.1768284, [735] := 2.257237, [736] := 2.213469, [737] := 3.8704424, [738] := 7.6158314, [739] := 13.024449, [740] := 19.277185, [741] := 26.336521, [742] := 32.726814, [743] := 40.680294, [744] := 49.146496, [745] := 57.794033, [746] := 66.491585, [747] := 72.91315, [748] := 80.466446, [749] := 87.25692, [750] := 93.06571, [751] := 96.44845, [752] := 99.33095, [753] := 100.844124, [754] := 101.03796, [755] := 100.33139, [756] := 98.36803, [757] := 95.56681, [758] := 92.07153, [759] := 88.1198, [760] := 84.03676, [761] := 78.75945, [762] := 72.806854, [763] := 66.31026, [764] := 60.5765, [765] := 52.673042, [766] := 44.88839, [767] := 36.45345, [768] := 28.387415, [769] := 22.797472, [770] := 16.032013, [771] := 10.173202, [772] := 6.3715367, [773] := 3.2264113, [774] := 2.0071268, [775] := 2.782467, [776] := 4.0892897, [777] := 8.409929, [778] := 11.961484, [779] := 17.951601, [780] := 25.41737,
        [781] := 32.80185, [782] := 40.64278, [783] := 47.408234, [784] := 56.44969, [785] := 64.953415, [786] := 73.06321, [787] := 79.04708, [788] := 85.85005, [789] := 91.64634, [790] := 96.26086, [791] := 99.32471, [792] := 100.68154, [793] := 101.10673, [794] := 100.3564, [795] := 98.50559, [796] := 96.42968, [797] := 93.14075, [798] := 88.957664, [799] := 84.349396, [800] := 84.349396);   // vector de potencia por comunicación
   VPotencia : REAL[1500] := ([0] := 5.9449345e-37, [1] := 5.9449345e-37, [2] := 5.9449345e-37, [3] := 5.9449345e-37, [4] := 5.9449345e-37, [5] := 5.9449345e-37, [6] := 5.9449345e-37, [7] := 5.9449345e-37, [8] := 5.9449345e-37, [9] := 5.9449345e-37, [10] := 5.9449345e-37, [11] := 5.9449345e-37, [12] := 5.9449345e-37, [13] := 5.9449345e-37, [14] := 5.9449345e-37, [15] := 5.9449345e-37, [16] := 5.9449345e-37, [17] := 5.9449345e-37, [18] := 5.9449345e-37, [19] := 5.9449345e-37, [20] := 5.9449345e-37, [21] := 5.9449345e-37, [22] := 5.9449345e-37, [23] := 5.9449345e-37, [24] := 5.9449345e-37, [25] := 5.9449345e-37, [26] := 5.9449345e-37, [27] := 5.9449345e-37, [28] := 5.9449345e-37, [29] := 5.9449345e-37, [30] := 5.9449345e-37, [31] := 5.9449345e-37, [32] := 5.9449345e-37, [33] := 5.9449345e-37, [34] := 5.9449345e-37, [35] := 5.9449345e-37, [36] := 5.9449345e-37, [37] := 5.9449345e-37, [38] := 5.9449345e-37, [39] := 5.9449345e-37, [40] := 5.9449345e-37, [41] := 5.9449345e-37, [42] := 5.9449345e-37, [43] := 5.9449345e-37, [44] := 5.9449345e-37, [45] := 5.9449345e-37, [46] := 5.9449345e-37, [47] := 5.9449345e-37, [48] := 5.9449345e-37, [49] := 5.9449345e-37, [50] := 5.9449345e-37, [51] := 5.9449345e-37, [52] := 5.9449345e-37, [53] := 5.9449345e-37, [54] := 5.9449345e-37, [55] := 5.9449345e-37, [56] := 5.9449345e-37, [57] := 5.9449345e-37, [58] := 5.9449345e-37, [59] := 5.9449345e-37,
        [60] := 5.9449345e-37, [61] := 5.9449345e-37, [62] := 5.9449345e-37, [63] := 5.9449345e-37, [64] := 5.9449345e-37, [65] := 5.9449345e-37, [66] := 5.9449345e-37, [67] := 5.9449345e-37, [68] := 5.9449345e-37, [69] := 5.9449345e-37, [70] := 5.9449345e-37, [71] := 5.9449345e-37, [72] := 5.9449345e-37, [73] := 5.9449345e-37, [74] := 5.9449345e-37, [75] := 5.9449345e-37, [76] := 5.9449345e-37, [77] := 5.9449345e-37, [78] := 5.9449345e-37, [79] := 5.9449345e-37, [80] := 5.9449345e-37, [81] := 5.9449345e-37, [82] := 5.9449345e-37, [83] := 5.9449345e-37, [84] := 5.9449345e-37, [85] := 5.9449345e-37, [86] := 5.9449345e-37, [87] := 5.9449345e-37, [88] := 5.9449345e-37, [89] := 5.9449345e-37, [90] := 5.9449345e-37, [91] := 5.9449345e-37, [92] := 5.9449345e-37, [93] := 5.9449345e-37, [94] := 5.9449345e-37, [95] := 5.9449345e-37, [96] := 5.9449345e-37, [97] := 5.9449345e-37, [98] := 5.9449345e-37, [99] := 5.9449345e-37, [100] := 5.9449345e-37, [101] := 5.9449345e-37, [102] := 5.9449345e-37, [103] := 5.9449345e-37, [104] := 5.9449345e-37, [105] := 5.9449345e-37, [106] := 5.9449345e-37, [107] := 5.9449345e-37, [108] := 5.9449345e-37, [109] := 5.9449345e-37, [110] := 5.9449345e-37, [111] := 5.9449345e-37, [112] := 5.9449345e-37, [113] := 5.9449345e-37, [114] := 5.9449345e-37, [115] := 5.9449345e-37, [116] := 5.9449345e-37, [117] := 5.9449345e-37, [118] := 5.9449345e-37, [119] := 5.9449345e-37,
        [120] := 5.9449345e-37, [121] := 5.9449345e-37, [122] := 5.9449345e-37, [123] := 5.9449345e-37, [124] := 5.9449345e-37, [125] := 5.9449345e-37, [126] := 5.9449345e-37, [127] := 5.9449345e-37, [128] := 5.9449345e-37, [129] := 5.9449345e-37, [130] := 5.9449345e-37, [131] := 5.9449345e-37, [132] := 5.9449345e-37, [133] := 5.9449345e-37, [134] := 5.9449345e-37, [135] := 5.9449345e-37, [136] := 5.9449345e-37, [137] := 5.9449345e-37, [138] := 5.9449345e-37, [139] := 5.9449345e-37, [140] := 5.9449345e-37, [141] := 5.9449345e-37, [142] := 5.9449345e-37, [143] := 5.9449345e-37, [144] := 5.9449345e-37, [145] := 5.9449345e-37, [146] := 5.9449345e-37, [147] := 5.9449345e-37, [148] := 5.9449345e-37, [149] := 5.9449345e-37, [150] := 5.9449345e-37, [151] := 5.9449345e-37, [152] := 5.9449345e-37, [153] := 5.9449345e-37, [154] := 5.9449345e-37, [155] := 5.9449345e-37, [156] := 5.9449345e-37, [157] := 5.9449345e-37, [158] := 5.9449345e-37, [159] := 5.9449345e-37, [160] := 5.9449345e-37, [161] := 5.9449345e-37, [162] := 5.9449345e-37, [163] := 5.9449345e-37, [164] := 5.9449345e-37, [165] := 5.9449345e-37, [166] := 5.9449345e-37, [167] := 5.9449345e-37, [168] := 5.9449345e-37, [169] := 5.9449345e-37, [170] := 5.9449345e-37, [171] := 5.9449345e-37, [172] := 5.9449345e-37, [173] := 5.9449345e-37, [174] := 5.9449345e-37, [175] := 5.9449345e-37, [176] := 5.9449345e-37, [177] := 5.9449345e-37, [178] := 5.9449345e-37, [179] := 5.9449345e-37,
        [180] := 5.9449345e-37, [181] := 5.9449345e-37, [182] := 5.9449345e-37, [183] := 5.9449345e-37, [184] := 5.9449345e-37, [185] := 5.9449345e-37, [186] := 5.9449345e-37, [187] := 5.9449345e-37, [188] := 5.9449345e-37, [189] := 5.9449345e-37, [190] := 5.9449345e-37, [191] := 5.9449345e-37, [192] := 5.9449345e-37, [193] := 5.9449345e-37, [194] := 5.9449345e-37, [195] := 5.9449345e-37, [196] := 5.9449345e-37, [197] := 5.9449345e-37, [198] := 5.9449345e-37, [199] := 5.9449345e-37, [200] := 5.9449345e-37, [201] := 5.9449345e-37, [202] := 5.9449345e-37, [203] := 5.9449345e-37, [204] := 5.9449345e-37, [205] := 5.9449345e-37, [206] := 5.9449345e-37, [207] := 5.9449345e-37, [208] := 5.9449345e-37, [209] := 5.9449345e-37, [210] := 5.9449345e-37, [211] := 5.9449345e-37, [212] := 5.9449345e-37, [213] := 5.9449345e-37, [214] := 5.9449345e-37, [215] := 5.9449345e-37, [216] := 5.9449345e-37, [217] := 5.9449345e-37, [218] := 5.9449345e-37, [219] := 5.9449345e-37, [220] := 5.9449345e-37, [221] := 5.9449345e-37, [222] := 5.9449345e-37, [223] := 5.9449345e-37, [224] := 5.9449345e-37, [225] := 5.9449345e-37, [226] := 5.9449345e-37, [227] := 5.9449345e-37, [228] := 5.9449345e-37, [229] := 5.9449345e-37, [230] := 5.9449345e-37, [231] := 5.9449345e-37, [232] := 5.9449345e-37, [233] := 5.9449345e-37, [234] := 5.9449345e-37, [235] := 5.9449345e-37, [236] := 5.9449345e-37, [237] := 5.9449345e-37, [238] := 5.9449345e-37, [239] := 5.9449345e-37,
        [240] := 5.9449345e-37, [241] := 5.9449345e-37, [242] := 5.9449345e-37, [243] := 5.9449345e-37, [244] := 5.9449345e-37, [245] := 5.9449345e-37, [246] := 5.9449345e-37, [247] := 5.9449345e-37, [248] := 5.9449345e-37, [249] := 5.9449345e-37, [250] := 5.9449345e-37, [251] := 5.9449345e-37, [252] := 5.9449345e-37, [253] := 5.9449345e-37, [254] := 5.9449345e-37, [255] := 5.9449345e-37, [256] := 5.9449345e-37, [257] := 5.9449345e-37, [258] := 5.9449345e-37, [259] := 5.9449345e-37, [260] := 5.9449345e-37, [261] := 5.9449345e-37, [262] := 5.9449345e-37, [263] := 5.9449345e-37, [264] := 5.9449345e-37, [265] := 5.9449345e-37, [266] := 5.9449345e-37, [267] := 5.9449345e-37, [268] := 5.9449345e-37, [269] := 5.9449345e-37, [270] := 5.9449345e-37, [271] := 5.9449345e-37, [272] := 5.9449345e-37, [273] := 5.9449345e-37, [274] := 5.9449345e-37, [275] := 5.9449345e-37, [276] := 5.9449345e-37, [277] := 5.9449345e-37, [278] := 5.9449345e-37, [279] := 5.9449345e-37, [280] := 5.9449345e-37, [281] := 5.9449345e-37, [282] := 5.9449345e-37, [283] := 5.9449345e-37, [284] := 5.9449345e-37, [285] := 5.9449345e-37, [286] := 5.9449345e-37, [287] := 5.9449345e-37, [288] := 5.9449345e-37, [289] := 5.9449345e-37, [290] := 5.9449345e-37, [291] := 5.9449345e-37, [292] := 5.9449345e-37, [293] := 5.9449345e-37, [294] := 5.9449345e-37, [295] := 5.9449345e-37, [296] := 5.9449345e-37, [297] := 5.9449345e-37, [298] := 5.9449345e-37, [299] := 5.9449345e-37,
        [300] := 5.9449345e-37, [301] := 5.9449345e-37, [302] := 5.9449345e-37, [303] := 5.9449345e-37, [304] := 5.9449345e-37, [305] := 5.9449345e-37, [306] := 5.9449345e-37, [307] := 5.9449345e-37, [308] := 5.9449345e-37, [309] := 5.9449345e-37, [310] := 5.9449345e-37, [311] := 5.9449345e-37, [312] := 5.9449345e-37, [313] := 5.9449345e-37, [314] := 5.9449345e-37, [315] := 5.9449345e-37, [316] := 5.9449345e-37, [317] := 5.9449345e-37, [318] := 5.9449345e-37, [319] := 5.9449345e-37, [320] := 5.9449345e-37, [321] := 5.9449345e-37, [322] := 5.9449345e-37, [323] := 5.9449345e-37, [324] := 5.9449345e-37, [325] := 5.9449345e-37, [326] := 5.9449345e-37, [327] := 5.9449345e-37, [328] := 5.9449345e-37, [329] := 5.9449345e-37, [330] := 5.9449345e-37, [331] := 5.9449345e-37, [332] := 5.9449345e-37, [333] := 5.9449345e-37, [334] := 5.9449345e-37, [335] := 5.9449345e-37, [336] := 5.9449345e-37, [337] := 5.9449345e-37, [338] := 5.9449345e-37, [339] := 5.9449345e-37, [340] := 5.9449345e-37, [341] := 5.9449345e-37, [342] := 5.9449345e-37, [343] := 5.9449345e-37, [344] := 5.9449345e-37, [345] := 5.9449345e-37, [346] := 5.9449345e-37, [347] := 5.9449345e-37, [348] := 5.9449345e-37, [349] := 5.9449345e-37, [350] := 5.9449345e-37, [351] := 5.9449345e-37, [352] := 5.9449345e-37, [353] := 5.9449345e-37, [354] := 5.9449345e-37, [355] := 5.9449345e-37, [356] := 5.9449345e-37, [357] := 5.9449345e-37, [358] := 5.9449345e-37, [359] := 5.9449345e-37,
        [360] := 5.9449345e-37, [361] := 5.9449345e-37, [362] := 5.9449345e-37, [363] := 5.9449345e-37, [364] := 5.9449345e-37, [365] := 5.9449345e-37, [366] := 5.9449345e-37, [367] := 5.9449345e-37, [368] := 5.9449345e-37, [369] := 5.9449345e-37, [370] := 5.9449345e-37, [371] := 5.9449345e-37, [372] := 5.9449345e-37, [373] := 5.9449345e-37, [374] := 5.9449345e-37, [375] := 5.9449345e-37, [376] := 5.9449345e-37, [377] := 5.9449345e-37, [378] := 5.9449345e-37, [379] := 5.9449345e-37, [380] := 5.9449345e-37, [381] := 5.9449345e-37, [382] := 5.9449345e-37, [383] := 5.9449345e-37, [384] := 5.9449345e-37, [385] := 5.9449345e-37, [386] := 5.9449345e-37, [387] := 5.9449345e-37, [388] := 5.9449345e-37, [389] := 5.9449345e-37, [390] := 5.9449345e-37, [391] := 5.9449345e-37, [392] := 5.9449345e-37, [393] := 5.9449345e-37, [394] := 5.9449345e-37, [395] := 5.9449345e-37, [396] := 5.9449345e-37, [397] := 5.9449345e-37, [398] := 5.9449345e-37, [399] := 5.9449345e-37, [400] := 5.9449345e-37, [401] := 5.9449345e-37, [402] := 5.9449345e-37, [403] := 5.9449345e-37, [404] := 5.9449345e-37, [405] := 5.9449345e-37, [406] := 5.9449345e-37, [407] := 5.9449345e-37, [408] := 5.9449345e-37, [409] := 5.9449345e-37, [410] := 5.9449345e-37, [411] := 5.9449345e-37, [412] := 5.9449345e-37, [413] := 5.9449345e-37, [414] := 5.9449345e-37, [415] := 5.9449345e-37, [416] := 5.9449345e-37, [417] := 5.9449345e-37, [418] := 5.9449345e-37, [419] := 5.9449345e-37,
        [420] := 5.9449345e-37, [421] := 5.9449345e-37, [422] := 5.9449345e-37, [423] := 5.9449345e-37, [424] := 5.9449345e-37, [425] := 5.9449345e-37, [426] := 5.9449345e-37, [427] := 5.9449345e-37, [428] := 5.9449345e-37, [429] := 5.9449345e-37, [430] := 5.9449345e-37, [431] := 5.9449345e-37, [432] := 5.9449345e-37, [433] := 5.9449345e-37, [434] := 5.9449345e-37, [435] := 5.9449345e-37, [436] := 5.9449345e-37, [437] := 5.9449345e-37, [438] := 5.9449345e-37, [439] := 5.9449345e-37, [440] := 5.9449345e-37, [441] := 5.9449345e-37, [442] := 5.9449345e-37, [443] := 5.9449345e-37, [444] := 5.9449345e-37, [445] := 5.9449345e-37, [446] := 5.9449345e-37, [447] := 5.9449345e-37, [448] := 5.9449345e-37, [449] := 5.9449345e-37, [450] := 5.9449345e-37, [451] := 5.9449345e-37, [452] := 5.9449345e-37, [453] := 5.9449345e-37, [454] := 5.9449345e-37, [455] := 5.9449345e-37, [456] := 5.9449345e-37, [457] := 5.9449345e-37, [458] := 5.9449345e-37, [459] := 5.9449345e-37, [460] := 5.9449345e-37, [461] := 5.9449345e-37, [462] := 5.9449345e-37, [463] := 5.9449345e-37, [464] := 5.9449345e-37, [465] := 5.9449345e-37, [466] := 5.9449345e-37, [467] := 5.9449345e-37, [468] := 5.9449345e-37, [469] := 5.9449345e-37, [470] := 5.9449345e-37, [471] := 5.9449345e-37, [472] := 5.9449345e-37, [473] := 5.9449345e-37, [474] := 5.9449345e-37, [475] := 5.9449345e-37, [476] := 5.9449345e-37, [477] := 5.9449345e-37, [478] := 5.9449345e-37, [479] := 5.9449345e-37,
        [480] := 5.9449345e-37, [481] := 5.9449345e-37, [482] := 5.9449345e-37, [483] := 5.9449345e-37, [484] := 5.9449345e-37, [485] := 5.9449345e-37, [486] := 5.9449345e-37, [487] := 5.9449345e-37, [488] := 5.9449345e-37, [489] := 5.9449345e-37, [490] := 5.9449345e-37, [491] := 5.9449345e-37, [492] := 5.9449345e-37, [493] := 5.9449345e-37, [494] := 5.9449345e-37, [495] := 5.9449345e-37, [496] := 5.9449345e-37, [497] := 5.9449345e-37, [498] := 5.9449345e-37, [499] := 5.9449345e-37, [500] := 5.9449345e-37, [501] := 5.9449345e-37, [502] := 5.9449345e-37, [503] := 5.9449345e-37, [504] := 5.9449345e-37, [505] := 5.9449345e-37, [506] := 5.9449345e-37, [507] := 5.9449345e-37, [508] := 5.9449345e-37, [509] := 5.9449345e-37, [510] := 5.9449345e-37, [511] := 5.9449345e-37, [512] := 5.9449345e-37, [513] := 5.9449345e-37, [514] := 5.9449345e-37, [515] := 5.9449345e-37, [516] := 5.9449345e-37, [517] := 5.9449345e-37, [518] := 5.9449345e-37, [519] := 5.9449345e-37, [520] := 5.9449345e-37, [521] := 5.9449345e-37, [522] := 5.9449345e-37, [523] := 5.9449345e-37, [524] := 5.9449345e-37, [525] := 5.9449345e-37, [526] := 5.9449345e-37, [527] := 5.9449345e-37, [528] := 5.9449345e-37, [529] := 5.9449345e-37, [530] := 5.9449345e-37, [531] := 5.9449345e-37, [532] := 5.9449345e-37, [533] := 5.9449345e-37, [534] := 5.9449345e-37, [535] := 5.9449345e-37, [536] := 5.9449345e-37, [537] := 5.9449345e-37, [538] := 5.9449345e-37, [539] := 5.9449345e-37,
        [540] := 5.9449345e-37, [541] := 5.9449345e-37, [542] := 5.9449345e-37, [543] := 5.9449345e-37, [544] := 5.9449345e-37, [545] := 5.9449345e-37, [546] := 5.9449345e-37, [547] := 5.9449345e-37, [548] := 5.9449345e-37, [549] := 5.9449345e-37, [550] := 5.9449345e-37, [551] := 5.9449345e-37, [552] := 5.9449345e-37, [553] := 5.9449345e-37, [554] := 5.9449345e-37, [555] := 5.9449345e-37, [556] := 5.9449345e-37, [557] := 5.9449345e-37, [558] := 5.9449345e-37, [559] := 5.9449345e-37, [560] := 5.9449345e-37, [561] := 5.9449345e-37, [562] := 5.9449345e-37, [563] := 5.9449345e-37, [564] := 5.9449345e-37, [565] := 5.9449345e-37, [566] := 5.9449345e-37, [567] := 5.9449345e-37, [568] := 5.9449345e-37, [569] := 5.9449345e-37, [570] := 5.9449345e-37, [571] := 5.9449345e-37, [572] := 5.9449345e-37, [573] := 5.9449345e-37, [574] := 5.9449345e-37, [575] := 5.9449345e-37, [576] := 5.9449345e-37, [577] := 5.9449345e-37, [578] := 5.9449345e-37, [579] := 5.9449345e-37, [580] := 5.9449345e-37, [581] := 5.9449345e-37, [582] := 5.9449345e-37, [583] := 5.9449345e-37, [584] := 5.9449345e-37, [585] := 5.9449345e-37, [586] := 5.9449345e-37, [587] := 5.9449345e-37, [588] := 5.9449345e-37, [589] := 5.9449345e-37, [590] := 5.9449345e-37, [591] := 5.9449345e-37, [592] := 5.9449345e-37, [593] := 5.9449345e-37, [594] := 5.9449345e-37, [595] := 5.9449345e-37, [596] := 5.9449345e-37, [597] := 5.9449345e-37, [598] := 5.9449345e-37, [599] := 5.9449345e-37,
        [600] := 5.9449345e-37, [601] := 5.9449345e-37, [602] := 5.9449345e-37, [603] := 5.9449345e-37, [604] := 5.9449345e-37, [605] := 5.9449345e-37, [606] := 5.9449345e-37, [607] := 5.9449345e-37, [608] := 5.9449345e-37, [609] := 5.9449345e-37, [610] := 5.9449345e-37, [611] := 5.9449345e-37, [612] := 5.9449345e-37, [613] := 5.9449345e-37, [614] := 5.9449345e-37, [615] := 5.9449345e-37, [616] := 5.9449345e-37, [617] := 5.9449345e-37, [618] := 5.9449345e-37, [619] := 5.9449345e-37, [620] := 5.9449345e-37, [621] := 5.9449345e-37, [622] := 5.9449345e-37, [623] := 5.9449345e-37, [624] := 5.9449345e-37, [625] := 5.9449345e-37, [626] := 5.9449345e-37, [627] := 5.9449345e-37, [628] := 5.9449345e-37, [629] := 5.9449345e-37, [630] := 5.9449345e-37, [631] := 5.9449345e-37, [632] := 5.9449345e-37, [633] := 5.9449345e-37, [634] := 5.9449345e-37, [635] := 5.9449345e-37, [636] := 5.9449345e-37, [637] := 5.9449345e-37, [638] := 5.9449345e-37, [639] := 5.9449345e-37, [640] := 5.9449345e-37, [641] := 5.9449345e-37, [642] := 5.9449345e-37, [643] := 5.9449345e-37, [644] := 5.9449345e-37, [645] := 5.9449345e-37, [646] := 5.9449345e-37, [647] := 5.9449345e-37, [648] := 5.9449345e-37, [649] := 5.9449345e-37, [650] := 5.9449345e-37, [651] := 5.9449345e-37, [652] := 5.9449345e-37, [653] := 5.9449345e-37, [654] := 5.9449345e-37, [655] := 5.9449345e-37, [656] := 5.9449345e-37, [657] := 5.9449345e-37, [658] := 5.9449345e-37, [659] := 5.9449345e-37,
        [660] := 5.9449345e-37, [661] := 5.9449345e-37, [662] := 5.9449345e-37, [663] := 5.9449345e-37, [664] := 5.9449345e-37, [665] := 5.9449345e-37, [666] := 5.9449345e-37, [667] := 5.9449345e-37, [668] := 5.9449345e-37, [669] := 5.9449345e-37, [670] := 5.9449345e-37, [671] := 5.9449345e-37, [672] := 5.9449345e-37, [673] := 5.9449345e-37, [674] := 5.9449345e-37, [675] := 5.9449345e-37, [676] := 5.9449345e-37, [677] := 5.9449345e-37, [678] := 5.9449345e-37, [679] := 5.9449345e-37, [680] := 5.9449345e-37, [681] := 5.9449345e-37, [682] := 5.9449345e-37, [683] := 5.9449345e-37, [684] := 5.9449345e-37, [685] := 5.9449345e-37, [686] := 5.9449345e-37, [687] := 5.9449345e-37, [688] := 5.9449345e-37, [689] := 5.9449345e-37, [690] := 5.9449345e-37, [691] := 5.9449345e-37, [692] := 5.9449345e-37, [693] := 5.9449345e-37, [694] := 5.9449345e-37, [695] := 5.9449345e-37, [696] := 5.9449345e-37, [697] := 5.9449345e-37, [698] := 5.9449345e-37, [699] := 5.9449345e-37, [700] := 5.9449345e-37, [701] := 5.9449345e-37, [702] := 5.9449345e-37, [703] := 5.9449345e-37, [704] := 5.9449345e-37, [705] := 5.9449345e-37, [706] := 5.9449345e-37, [707] := 5.9449345e-37, [708] := 5.9449345e-37, [709] := 5.9449345e-37, [710] := 5.9449345e-37, [711] := 5.9449345e-37, [712] := 5.9449345e-37, [713] := 5.9449345e-37, [714] := 5.9449345e-37, [715] := 5.9449345e-37, [716] := 5.9449345e-37, [717] := 5.9449345e-37, [718] := 5.9449345e-37, [719] := 5.9449345e-37,
        [720] := 5.9449345e-37, [721] := 5.9449345e-37, [722] := 5.9449345e-37, [723] := 5.9449345e-37, [724] := 5.9449345e-37, [725] := 5.9449345e-37, [726] := 5.9449345e-37, [727] := 5.9449345e-37, [728] := 5.9449345e-37, [729] := 5.9449345e-37, [730] := 5.9449345e-37, [731] := 5.9449345e-37, [732] := 5.9449345e-37, [733] := 5.9449345e-37, [734] := 5.9449345e-37, [735] := 5.9449345e-37, [736] := 5.9449345e-37, [737] := 5.9449345e-37, [738] := 5.9449345e-37, [739] := 5.9449345e-37, [740] := 5.9449345e-37, [741] := 5.9449345e-37, [742] := 5.9449345e-37, [743] := 5.9449345e-37, [744] := 5.9449345e-37, [745] := 5.9449345e-37, [746] := 5.9449345e-37, [747] := 5.9449345e-37, [748] := 5.9449345e-37, [749] := 5.9449345e-37, [750] := 5.9449345e-37, [751] := 5.9449345e-37, [752] := 5.9449345e-37, [753] := 5.9449345e-37, [754] := 5.9449345e-37, [755] := 5.9449345e-37, [756] := 5.9449345e-37, [757] := 5.9449345e-37, [758] := 5.9449345e-37, [759] := 5.9449345e-37, [760] := 5.9449345e-37, [761] := 5.9449345e-37, [762] := 5.9449345e-37, [763] := 5.9449345e-37, [764] := 5.9449345e-37, [765] := 5.9449345e-37, [766] := 5.9449345e-37, [767] := 5.9449345e-37, [768] := 5.9449345e-37, [769] := 5.9449345e-37, [770] := 5.9449345e-37, [771] := 5.9449345e-37, [772] := 5.9449345e-37, [773] := 5.9449345e-37, [774] := 5.9449345e-37, [775] := 5.9449345e-37, [776] := 5.9449345e-37, [777] := 5.9449345e-37, [778] := 5.9449345e-37, [779] := 5.9449345e-37,
        [780] := 5.9449345e-37, [781] := 5.9449345e-37, [782] := 5.9449345e-37, [783] := 5.9449345e-37, [784] := 5.9449345e-37, [785] := 5.9449345e-37, [786] := 5.9449345e-37, [787] := 5.9449345e-37, [788] := 5.9449345e-37, [789] := 5.9449345e-37, [790] := 5.9449345e-37, [791] := 5.9449345e-37, [792] := 5.9449345e-37, [793] := 5.9449345e-37, [794] := 5.9449345e-37, [795] := 5.9449345e-37, [796] := 5.9449345e-37, [797] := 5.9449345e-37, [798] := 5.9449345e-37, [799] := 5.9449345e-37, [800] := 5.9449345e-37);
   VPotenciaC : REAL[1500] := ([1] := -5.9576063, [2] := -5.9576063, [3] := -5.9576063, [4] := -5.9576063, [5] := -5.9576063, [6] := -5.9576063, [7] := -5.9576063, [8] := -5.9576063, [9] := -5.9576063, [10] := -5.9576063, [11] := -5.9576063, [12] := -5.9576063, [13] := -5.9576063, [14] := -5.9576063, [15] := -5.9576063, [16] := -5.9576063, [17] := -5.9576063, [18] := -5.9576063, [19] := -5.9576063, [20] := -5.9576063, [21] := -5.9576063, [22] := -5.9576063, [23] := -5.9576063, [24] := -5.9576063, [25] := -5.9576063, [26] := -5.9576063, [27] := -5.9576063, [28] := -5.9576063, [29] := -5.9576063, [30] := -5.9576063, [31] := -5.9576063, [32] := -5.9576063, [33] := -5.9576063, [34] := -5.9576063, [35] := -5.9576063, [36] := -5.9576063, [37] := -5.9576063, [38] := -5.9576063, [39] := -5.9576063, [40] := -5.9576063, [41] := -5.9576063, [42] := -5.9576063, [43] := -5.9576063, [44] := -5.9576063, [45] := -5.9576063, [46] := -5.9576063, [47] := -5.9576063, [48] := -5.9576063, [49] := -5.9576063, [50] := -5.9576063, [51] := -5.9576063, [52] := -5.9576063, [53] := -5.9576063, [54] := -5.9576063, [55] := -5.9576063, [56] := -5.9576063, [57] := -5.9576063, [58] := -5.9576063, [59] := -5.9576063, [60] := -5.9576063,
        [61] := -5.9576063, [62] := -5.9576063, [63] := -5.9576063, [64] := -5.9576063, [65] := -5.9576063, [66] := -5.9576063, [67] := -5.9576063, [68] := -5.9576063, [69] := -5.9576063, [70] := -5.9576063, [71] := -5.9576063, [72] := -5.9576063, [73] := -5.9576063, [74] := -5.9576063, [75] := -5.9576063, [76] := -5.9576063, [77] := -5.9576063, [78] := -5.9576063, [79] := -5.9576063, [80] := -5.9576063, [81] := -5.9576063, [82] := -5.9576063, [83] := -5.9576063, [84] := -5.9576063, [85] := -5.9576063, [86] := -5.9576063, [87] := -5.9576063, [88] := -5.9576063, [89] := -5.9576063, [90] := -5.9576063, [91] := -5.9576063, [92] := -5.9576063, [93] := -5.9576063, [94] := -5.9576063, [95] := -5.9576063, [96] := -5.9576063, [97] := -5.9576063, [98] := -5.9576063, [99] := -5.9576063, [100] := -5.9576063, [101] := -5.9576063, [102] := -5.9576063, [103] := -5.9576063, [104] := -5.9576063, [105] := -5.9576063, [106] := -5.9576063, [107] := -5.9576063, [108] := -5.9576063, [109] := -5.9576063, [110] := -5.9576063, [111] := -5.9576063, [112] := -5.9576063, [113] := -5.9576063, [114] := -5.9576063, [115] := -5.9576063, [116] := -5.9576063, [117] := -5.9576063, [118] := -5.9576063, [119] := -5.9576063, [120] := -5.9576063,
        [121] := -5.9576063, [122] := -5.9576063, [123] := -5.9576063, [124] := -5.9576063, [125] := -5.9576063, [126] := -5.9576063, [127] := -5.9576063, [128] := -5.9576063, [129] := -5.9576063, [130] := -5.9576063, [131] := -5.9576063, [132] := -5.9576063, [133] := -5.9576063, [134] := -5.9576063, [135] := -5.9576063, [136] := -5.9576063, [137] := -5.9576063, [138] := -5.9576063, [139] := -5.9576063, [140] := -5.9576063, [141] := -5.9576063, [142] := -5.9576063, [143] := -5.9576063, [144] := -5.9576063, [145] := -5.9576063, [146] := -5.9576063, [147] := -5.9576063, [148] := -5.9576063, [149] := -5.9576063, [150] := -5.9576063, [151] := -5.9576063, [152] := -5.9576063, [153] := -5.9576063, [154] := -5.9576063, [155] := -5.9576063, [156] := -5.9576063, [157] := -5.9576063, [158] := -5.9576063, [159] := -5.9576063, [160] := -5.9576063, [161] := -5.9576063, [162] := -5.9576063, [163] := -5.9576063, [164] := -5.9576063, [165] := -5.9576063, [166] := -5.9576063, [167] := -5.9576063, [168] := -5.9576063, [169] := -5.9576063, [170] := -5.9576063, [171] := -5.9576063, [172] := -5.9576063, [173] := -5.9576063, [174] := -5.9576063, [175] := -5.9576063, [176] := -5.9576063, [177] := -5.9576063, [178] := -5.9576063, [179] := -5.9576063, [180] := -5.9576063,
        [181] := -5.9576063, [182] := -5.9576063, [183] := -5.9576063, [184] := -5.9576063, [185] := -5.9576063, [186] := -5.9576063, [187] := -5.9576063, [188] := -5.9576063, [189] := -5.9576063, [190] := -5.9576063, [191] := -5.9576063, [192] := -5.9576063, [193] := -5.9576063, [194] := -5.9576063, [195] := -5.9576063, [196] := -5.9576063, [197] := -5.9576063, [198] := -5.9576063, [199] := -5.9576063, [200] := -5.9576063, [201] := -5.9576063, [202] := -5.9576063, [203] := -5.9576063, [204] := -5.9576063, [205] := -5.9576063, [206] := -5.9576063, [207] := -5.9576063, [208] := -5.9576063, [209] := -5.9576063, [210] := -5.9576063, [211] := -5.9576063, [212] := -5.9576063, [213] := -5.9576063, [214] := -5.9576063, [215] := -5.9576063, [216] := -5.9576063, [217] := -5.9576063, [218] := -5.9576063, [219] := -5.9576063, [220] := -5.9576063, [221] := -5.9576063, [222] := -5.9576063, [223] := -5.9576063, [224] := -5.9576063, [225] := -5.9576063, [226] := -5.9576063, [227] := -5.9576063, [228] := -5.9576063, [229] := -5.9576063, [230] := -5.9576063, [231] := -5.9576063, [232] := -5.9576063, [233] := -5.9576063, [234] := -5.9576063, [235] := -5.9576063, [236] := -5.9576063, [237] := -5.9576063, [238] := -5.9576063, [239] := -5.9576063, [240] := -5.9576063,
        [241] := -5.9576063, [242] := -5.9576063, [243] := -5.9576063, [244] := -5.9576063, [245] := -5.9576063, [246] := -5.9576063, [247] := -5.9576063, [248] := -5.9576063, [249] := -5.9576063, [250] := -5.9576063, [251] := -5.9576063, [252] := -5.9576063, [253] := -5.9576063, [254] := -5.9576063, [255] := -5.9576063, [256] := -5.9576063, [257] := -5.9576063, [258] := -5.9576063, [259] := -5.9576063, [260] := -5.9576063, [261] := -5.9576063, [262] := -5.9576063, [263] := -5.9576063, [264] := -5.9576063, [265] := -5.9576063, [266] := -5.9576063, [267] := -5.9576063, [268] := -5.9576063, [269] := -5.9576063, [270] := -5.9576063, [271] := -5.9576063, [272] := -5.9576063, [273] := -5.9576063, [274] := -5.9576063, [275] := -5.9576063, [276] := -5.9576063, [277] := -5.9576063, [278] := -5.9576063, [279] := -5.9576063, [280] := -5.9576063, [281] := -5.9576063, [282] := -5.9576063, [283] := -5.9576063, [284] := -5.9576063, [285] := -5.9576063, [286] := -5.9576063, [287] := -5.9576063, [288] := -5.9576063, [289] := -5.9576063, [290] := -5.9576063, [291] := -5.9576063, [292] := -5.9576063, [293] := -5.9576063, [294] := -5.9576063, [295] := -5.9576063, [296] := -5.9576063, [297] := -5.9576063, [298] := -5.9576063, [299] := -5.9576063, [300] := -5.9576063,
        [301] := -5.9576063, [302] := -5.9576063, [303] := -5.9576063, [304] := -5.9576063, [305] := -5.9576063, [306] := -5.9576063, [307] := -5.9576063, [308] := -5.9576063, [309] := -5.9576063, [310] := -5.9576063, [311] := -5.9576063, [312] := -5.9576063, [313] := -5.9576063, [314] := -5.9576063, [315] := -5.9576063, [316] := -5.9576063, [317] := -5.9576063, [318] := -5.9576063, [319] := -5.9576063, [320] := -5.9576063, [321] := -5.9576063, [322] := -5.9576063, [323] := -5.9576063, [324] := -5.9576063, [325] := -5.9576063, [326] := -5.9576063, [327] := -5.9576063, [328] := -5.9576063, [329] := -5.9576063, [330] := -5.9576063, [331] := -5.9576063, [332] := -5.9576063, [333] := -5.9576063, [334] := -5.9576063, [335] := -5.9576063, [336] := -5.9576063, [337] := -5.9576063, [338] := -5.9576063, [339] := -5.9576063, [340] := -5.9576063, [341] := -5.9576063, [342] := -5.9576063, [343] := -5.9576063, [344] := -5.9576063, [345] := -5.9576063, [346] := -5.9576063, [347] := -5.9576063, [348] := -5.9576063, [349] := -5.9576063, [350] := -5.9576063, [351] := -5.9576063, [352] := -5.9576063, [353] := -5.9576063, [354] := -5.9576063, [355] := -5.9576063, [356] := -5.9576063, [357] := -5.9576063, [358] := -5.9576063, [359] := -5.9576063, [360] := -5.9576063,
        [361] := -5.9576063, [362] := -5.9576063, [363] := -5.9576063, [364] := -5.9576063, [365] := -5.9576063, [366] := -5.9576063, [367] := -5.9576063, [368] := -5.9576063, [369] := -5.9576063, [370] := -5.9576063, [371] := -5.9576063, [372] := -5.9576063, [373] := -5.9576063, [374] := -5.9576063, [375] := -5.9576063, [376] := -5.9576063, [377] := -5.9576063, [378] := -5.9576063, [379] := -5.9576063, [380] := -5.9576063, [381] := -5.9576063, [382] := -5.9576063, [383] := -5.9576063, [384] := -5.9576063, [385] := -5.9576063, [386] := -5.9576063, [387] := -5.9576063, [388] := -5.9576063, [389] := -5.9576063, [390] := -5.9576063, [391] := -5.9576063, [392] := -5.9576063, [393] := -5.9576063, [394] := -5.9576063, [395] := -5.9576063, [396] := -5.9576063, [397] := -5.9576063, [398] := -5.9576063, [399] := -5.9576063, [400] := -5.9576063, [401] := -5.9576063, [402] := -5.9576063, [403] := -5.9576063, [404] := -5.9576063, [405] := -5.9576063, [406] := -5.9576063, [407] := -5.9576063, [408] := -5.9576063, [409] := -5.9576063, [410] := -5.9576063, [411] := -5.9576063, [412] := -5.9576063, [413] := -5.9576063, [414] := -5.9576063, [415] := -5.9576063, [416] := -5.9576063, [417] := -5.9576063, [418] := -5.9576063, [419] := -5.9576063, [420] := -5.9576063,
        [421] := -5.9576063, [422] := -5.9576063, [423] := -5.9576063, [424] := -5.9576063, [425] := -5.9576063, [426] := -5.9576063, [427] := -5.9576063, [428] := -5.9576063, [429] := -5.9576063, [430] := -5.9576063, [431] := -5.9576063, [432] := -5.9576063, [433] := -5.9576063, [434] := -5.9576063, [435] := -5.9576063, [436] := -5.9576063, [437] := -5.9576063, [438] := -5.9576063, [439] := -5.9576063, [440] := -5.9576063, [441] := -5.9576063, [442] := -5.9576063, [443] := -5.9576063, [444] := -5.9576063, [445] := -5.9576063, [446] := -5.9576063, [447] := -5.9576063, [448] := -5.9576063, [449] := -5.9576063, [450] := -5.9576063, [451] := -5.9576063, [452] := -5.9576063, [453] := -5.9576063, [454] := -5.9576063, [455] := -5.9576063, [456] := -5.9576063, [457] := -5.9576063, [458] := -5.9576063, [459] := -5.9576063, [460] := -5.9576063, [461] := -5.9576063, [462] := -5.9576063, [463] := -5.9576063, [464] := -5.9576063, [465] := -5.9576063, [466] := -5.9576063, [467] := -5.9576063, [468] := -5.9576063, [469] := -5.9576063, [470] := -5.9576063, [471] := -5.9576063, [472] := -5.9576063, [473] := -5.9576063, [474] := -5.9576063, [475] := -5.9576063, [476] := -5.9576063, [477] := -5.9576063, [478] := -5.9576063, [479] := -5.9576063, [480] := -5.9576063,
        [481] := -5.9576063, [482] := -5.9576063, [483] := -5.9576063, [484] := -5.9576063, [485] := -5.9576063, [486] := -5.9576063, [487] := -5.9576063, [488] := -5.9576063, [489] := -5.9576063, [490] := -5.9576063, [491] := -5.9576063, [492] := -5.9576063, [493] := -5.9576063, [494] := -5.9576063, [495] := -5.9576063, [496] := -5.9576063, [497] := -5.9576063, [498] := -5.9576063, [499] := -5.9576063, [500] := -5.9576063, [501] := -5.9576063, [502] := -5.9576063, [503] := -5.9576063, [504] := -5.9576063, [505] := -5.9576063, [506] := -5.9576063, [507] := -5.9576063, [508] := -5.9576063, [509] := -5.9576063, [510] := -5.9576063, [511] := -5.9576063, [512] := -5.9576063, [513] := -5.9576063, [514] := -5.9576063, [515] := -5.9576063, [516] := -5.9576063, [517] := -5.9576063, [518] := -5.9576063, [519] := -5.9576063, [520] := -5.9576063, [521] := -5.9576063, [522] := -5.9576063, [523] := -5.9576063, [524] := -5.9576063, [525] := -5.9576063, [526] := -5.9576063, [527] := -5.9576063, [528] := -5.9576063, [529] := -5.9576063, [530] := -5.9576063, [531] := -5.9576063, [532] := -5.9576063, [533] := -5.9576063, [534] := -5.9576063, [535] := -5.9576063, [536] := -5.9576063, [537] := -5.9576063, [538] := -5.9576063, [539] := -5.9576063, [540] := -5.9576063,
        [541] := -5.9576063, [542] := -5.9576063, [543] := -5.9576063, [544] := -5.9576063, [545] := -5.9576063, [546] := -5.9576063, [547] := -5.9576063, [548] := -5.9576063, [549] := -5.9576063, [550] := -5.9576063, [551] := -5.9576063, [552] := -5.9576063, [553] := -5.9576063, [554] := -5.9576063, [555] := -5.9576063, [556] := -5.9576063, [557] := -5.9576063, [558] := -5.9576063, [559] := -5.9576063, [560] := -5.9576063, [561] := -5.9576063, [562] := -5.9576063, [563] := -5.9576063, [564] := -5.9576063, [565] := -5.9576063, [566] := -5.9576063, [567] := -5.9576063, [568] := -5.9576063, [569] := -5.9576063, [570] := -5.9576063, [571] := -5.9576063, [572] := -5.9576063, [573] := -5.9576063, [574] := -5.9576063, [575] := -5.9576063, [576] := -5.9576063, [577] := -5.9576063, [578] := -5.9576063, [579] := -5.9576063, [580] := -5.9576063, [581] := -5.9576063, [582] := -5.9576063, [583] := -5.9576063, [584] := -5.9576063, [585] := -5.9576063, [586] := -5.9576063, [587] := -5.9576063, [588] := -5.9576063, [589] := -5.9576063, [590] := -5.9576063, [591] := -5.9576063, [592] := -5.9576063, [593] := -5.9576063, [594] := -5.9576063, [595] := -5.9576063, [596] := -5.9576063, [597] := -5.9576063, [598] := -5.9576063, [599] := -5.9576063, [600] := -5.9576063,
        [601] := -5.9576063, [602] := -5.9576063, [603] := -5.9576063, [604] := -5.9576063, [605] := -5.9576063, [606] := -5.9576063, [607] := -5.9576063, [608] := -5.9576063, [609] := -5.9576063, [610] := -5.9576063, [611] := -5.9576063, [612] := -5.9576063, [613] := -5.9576063, [614] := -5.9576063, [615] := -5.9576063, [616] := -5.9576063, [617] := -5.9576063, [618] := -5.9576063, [619] := -5.9576063, [620] := -5.9576063, [621] := -5.9576063, [622] := -5.9576063, [623] := -5.9576063, [624] := -5.9576063, [625] := -5.9576063, [626] := -5.9576063, [627] := -5.9576063, [628] := -5.9576063, [629] := -5.9576063, [630] := -5.9576063, [631] := -5.9576063, [632] := -5.9576063, [633] := -5.9576063, [634] := -5.9576063, [635] := -5.9576063, [636] := -5.9576063, [637] := -5.9576063, [638] := -5.9576063, [639] := -5.9576063, [640] := -5.9576063, [641] := -5.9576063, [642] := -5.9576063, [643] := -5.9576063, [644] := -5.9576063, [645] := -5.9576063, [646] := -5.9576063, [647] := -5.9576063, [648] := -5.9576063, [649] := -5.9576063, [650] := -5.9576063, [651] := -5.9576063, [652] := -5.9576063, [653] := -5.9576063, [654] := -5.9576063, [655] := -5.9576063, [656] := -5.9576063, [657] := -5.9576063, [658] := -5.9576063, [659] := -5.9576063, [660] := -5.9576063,
        [661] := -5.9576063, [662] := -5.9576063, [663] := -5.9576063, [664] := -5.9576063, [665] := -5.9576063, [666] := -5.9576063, [667] := -5.9576063, [668] := -5.9576063, [669] := -5.9576063, [670] := -5.9576063, [671] := -5.9576063, [672] := -5.9576063, [673] := -5.9576063, [674] := -5.9576063, [675] := -5.9576063, [676] := -5.9576063, [677] := -5.9576063, [678] := -5.9576063, [679] := -5.9576063, [680] := -5.9576063, [681] := -5.9576063, [682] := -5.9576063, [683] := -5.9576063, [684] := -5.9576063, [685] := -5.9576063, [686] := -5.9576063, [687] := -5.9576063, [688] := -5.9576063, [689] := -5.9576063, [690] := -5.9576063, [691] := -5.9576063, [692] := -5.9576063, [693] := -5.9576063);   // Vector de potencia cableado
   VProximetro : BOOL[1504] := ([0] := 1);
END_VAR
